						IF GradientToggle THEN
							st_LEDControl.Execute := FALSE;
							SFCStep := 4;
						END_IF
						GradientToggle := NOT GradientToggle;
					END_IF
					
				3: 
					IF NOT animationReady AND NOT LedBusy.Q THEN
							AnimationReady := SetAnimation(ActiveLeds := ui_activeLeds, charging:= getChargingState() = eDCstate.charging, reset := getChargingState() = eDCstate.idle, ledstoAnimate := LedsToAnimate);
					END_IF
					
					IF AnimationReady THEN
						AnimationReady := FALSE;
						st_LEDControl.Execute := NOT st_LEDControl.Execute;
						SFCStep := SFCStep + 1;
					END_IF
				ELSE
					bufferReady := TRUE;
			END_CASE
			
			ton_LEDdataSend(in:= NOT ton_LEDdataSend.Q AND bufferReady);
			IF ton_LEDDataSend.Q THEN
				ReadyToTransmit := TRUE;
			END_IF
			
			IF ReadyToTransmit AND NOT ledbusy.Q THEN
				SFCStep := 0;
				st_LEDControl.UPDATE 	:= NOT st_LEDControl.UPDATE;
				st_LEDControl.Execute 	:= NOT st_LEDControl.execute;	
			END_IF		
	END_CASE
END_IF

METHOD GetChargingState : eDCstate; 
VAR_INPUT
END_VAR
IF machinedata.r_DCCurrent > 10 THEN
	GetChargingState := eDCstate.discharging;
	//b_charging := FALSE;	
	//b_discharging := TRUE;
ELSIF machinedata.r_DCCurrent < -10 THEN
	GetChargingState := eDCstate.charging;
	//b_charging := TRUE;
	//b_discharging := FALSE;
ELSE
	GetChargingState := eDCstate.idle;
	//b_discharging := FALSE;
	//b_charging := FALSE;	
END_IF
END_METHOD

METHOD SetAnimation : BOOL;
VAR_INPUT
	ActiveLeds			: UINT;
	Charging			: BOOL;
	reset				: BOOL;
	LedsToAnimate		: BYTE := 5;	
END_VAR

VAR_INST
	AnimateResetToggle	: BYTE;
	//moveCounter			: CTUD;
	//ready				: BOOL;
	ledcounter			: BYTE;
END_VAR

//movecounter(pv := LedsToAnimate +1);
//moveCounter.LOAD := moveCounter.QD AND Charging;
//moveCounter.Reset := moveCounter.CV > movecounter.PV AND NOT Charging OR Reset;

//CASE AnimateResetToggle OF
//0:		AnimateResetToggle := AnimateResetToggle +1;
//		moveCounter.CU := FALSE;
//		moveCounter.CD := FALSE;
//	ELSE
//		AnimateResetToggle := 0;
//		moveCounter.cu := NOT charging;
//		movecounter.cd := Charging;
//		st_LEDControl.length 	:= 1;
//		st_LEDControl.command	:= 1; //move
//		st_LEDControl.parameter := 0;
//		st_LEDControl.index :=  ui_ActiveLeds + moveCounter.CV -1;
//		SetAnimation := TRUE;
//END_CASE

IF NOT RESET THEN
	ledcounter := ledcounter + SEL(charging,1 ,-1);
	IF ledcounter >= LedsToAnimate * 2 OR ledcounter = 0 THEN
		ledcounter := SEL(charging,0 ,LedsToAnimate * 2);	 
	END_IF
	
	st_LEDControl.length 	:= 1;
	st_LEDControl.command	:= 1; //move
	st_LEDControl.parameter := 
	st_LEDControl.index :=  ActiveLeds + ledcounter/2;
ELSE
	ledcounter := 0;
END_IF

SetAnimation := TRUE;
END_METHOD

METHOD SetColor : LEDColor

VAR_INPUT
	Brightness		: BYTE;
END_VAR

VAR
	tempColorValue	: USINT;
END_VAR
CASE machinedata.e_systemStatus OF
	eSystemStatus.neutral: 		
		SetColor.blue	:= Brightness;
		SetColor.red	:= Brightness;
		SetColor.green	:= Brightness;

	eSystemStatus.normal: 
		SetColor.blue	:= 0;
		SetColor.red	:= 0;
		SetColor.green	:= Brightness;
	
	eSystemStatus.attention: 
		SetColor.blue	:= Brightness;
		SetColor.red	:= 0;
		SetColor.green	:= 0;
	eSystemStatus.warning: //yelow
		SetColor.blue	:= 0;
		SetColor.red	:= Brightness;
		SetColor.green	:= Brightness/3;
	
	eSystemStatus.error: 
		SetColor.blue	:= 0;
		SetColor.red	:= Brightness;
		SetColor.green	:= 0;	
END_CASE

//Change RGB order
IF st_params.ColorOrder = eColorOrder.GRB THEN
	tempColorValue := setColor.Red;
	setcolor.red := setcolor.green;
	SetColor.green := tempColorValue;
END_IF
END_METHOD

END_FUNCTION_BLOCK

// ---- POUs/Objects/Enclosure/Climate/FB_EnclosureClimate.TcPOU
FUNCTION_BLOCK FB_EnclosureClimate
VAR_IN_OUT CONSTANT
	st_params				: ST_EnclosureClimate_params;
END_VAR
VAR_OUTPUT
	get						: ST_EnclosureClimate_get;
END_VAR

VAR
	TempRead		AT %I* : ST_AnalogInputData;
	HumRead			AT %I* : ST_AnalogInputData;
	
	scaleTemp				: FB_CTRL_SCALE;
	scaleHum				: FB_CTRL_SCALE;
	scaleParams				: ST_CTRL_SCALE_Params;
END_VAR

scaleParams.tCtrlCycleTime := T#100MS;
	scaleParams.tTaskCycleTime := T#1MS;
	scaleParams.fInMax := 16#7FFF;
	scaleParams.fInMin := 16#0000;
	scaleParams.fOutMax := 60;
	scaleParams.fOutMin:= -40;

scaleTemp(fin := TempRead.Value, fout => get.r_Temperature, stParams := scaleParams);
scaleParams.fOutMax := 100;
scaleParams.fOutMin := 0;
scaleHum(fin := HumRead.Value, fout => get.r_Humidity, stParams := scaleParams);

METHOD PUBLIC GetDiagnostics
VAR_IN_OUT
	AddError		: ARRAY [*] OF FB_AddErrorST;
	a_ActiveEvents	: ARRAY [*] OF ST_ErrorStruct;
	w_Index			: WORD;
END_VAR


VAR
	by_errCt	: BYTE;
	by_warnCt	: BYTE;
END_VAR
	(*Humidity High*)		AddError[w_Index](
		b_ErrorTrig			:= get.events.b_HumidityHigh,
		out_ST_Error			:= a_ActiveEvents[w_Index],
		w_ErrorID					:= 1,
		e_ObjectID				:=  eObject_ID.Enclosure_climate,
		s_Message				:= 'humidity high',
		e_sev					:= eseverity.Warning,
		b_AutoClear			:= TRUE
		);
		w_Index := w_Index +1;
	
	(*Humidity Too High*)		AddError[w_Index](
		b_ErrorTrig			:= get.events.b_HumidityTooHigh,
		out_ST_Error			:= a_ActiveEvents[w_Index],
		w_ErrorID					:= 2,
		s_Message				:= 'humidity too high',
		e_sev					:= eseverity.QuickShutdown,
		e_ErrAckAccess		:= eErrAckAccess.Operator
	);
	w_Index := w_Index +1;
	
	(*Temperature High*)		AddError[w_Index](
		b_ErrorTrig			:= get.events.b_TemperatureHigh,
		out_ST_Error			:= a_ActiveEvents[w_Index],
		w_ErrorID					:= 3,
		s_Message				:= 'temperature high',
		e_sev					:= eseverity.warning,
		b_AutoClear			:= TRUE
	);
	w_Index := w_Index +1;
	
	(*Temperature Too High*)	AddError[w_Index](
		b_ErrorTrig			:= get.events.b_TemperatureTooHigh,
		out_ST_Error			:= a_ActiveEvents[w_Index],
		w_ErrorID					:= 4,
		s_Message				:= 'temperature too high',
		e_sev					:= eseverity.Quickshutdown,
		e_ErrAckAccess		:= eErrAckAccess.Operator
	);

	w_Index := w_Index +1;
	
	(*Temperature Low*)	AddError[w_Index](
		b_ErrorTrig			:= get.events.b_TemperatureLow,
		out_ST_Error			:= a_ActiveEvents[w_Index],
		w_ErrorID					:= 5,
		s_Message				:= 'temperature low',
		e_sev					:= eseverity.Warning,
		b_AutoClear			:= TRUE
	);
	w_Index := w_Index +1;
	
	(*Temperature Too Low*)	AddError[w_Index](
		b_ErrorTrig			:= get.events.b_TemperatureTooLow,
		out_ST_Error			:= a_ActiveEvents[w_Index],
		w_ErrorID					:= 6,
		s_Message				:= 'temperature too low',
		e_sev					:= eseverity.Normalshutdown,
		e_ErrAckAccess		:= eErrAckAccess.Operator
	);
	w_Index := w_Index +1;
	
	(*4-20ma Overrange*)	AddError[w_Index](
		b_ErrorTrig			:= get.events.b_AIOverrange,
		out_ST_Error			:= a_ActiveEvents[w_Index],
		w_ErrorID					:= 7,
		s_Message				:= 'analog input temp/humid overrange',
		e_sev					:= eseverity.Warning,
		b_AutoClear			:= TRUE
	);
	w_Index := w_Index +1;
	
	(*4-20ma Underrange*)	AddError[w_Index](
		b_ErrorTrig			:= get.events.b_AIUnderrange,
		out_ST_Error			:= a_ActiveEvents[w_Index],
		w_ErrorID					:= 8,
		s_Message				:= 'analog input temp/humid underrange',
		e_sev					:= eseverity.Warning,
		b_AutoClear			:= TRUE
	);
	w_Index := w_Index +1;
	
	(*Analog input error*)	AddError[w_Index](
		b_ErrorTrig			:= get.events.b_AIError,
		out_ST_Error			:= a_ActiveEvents[w_Index],
		w_ErrorID					:= 9,
		s_Message				:= 'analog input temp/humid error',
		e_sev					:= eseverity.warning,
		b_AutoClear			:= TRUE
	);
	w_Index := w_Index +1;
	
	(*Analog input error*)	AddError[w_Index](
		b_ErrorTrig				:= get.events.b_DewpointTooHigh,
		out_ST_Error			:= a_ActiveEvents[w_Index],
		w_ErrorID				:= 10,
		s_Message				:= 'dewpoint too high alarm',
		e_sev					:= eseverity.normalshutdown,
	);
	w_Index := w_Index +1;
END_METHOD

METHOD PRIVATE SetEvents : BOOL
VAR_IN_OUT
	get : ST_EnclosureClimate_get;
	st_params : ST_EnclosureClimate_params;
END_VAR

VAR_INST
	sr_HumHigh			: SR;
	sr_HumTooHigh		: SR;
	sr_TempHigh			: SR;
	sr_TempTooHigh		: SR;
	sr_TempLow			: SR;
	sr_TempTooLow		: SR;
END_VAR
//set events
get.events.b_AIError := TempRead.Status.Error OR HumRead.Status.Error;
get.events.b_AIUnderrange := TempRead.Status.Underrange OR HumRead.Status.Underrange;
get.events.b_AIOverrange := TempRead.Status.Overrange OR HumRead.Status.Overrange;

sr_HumHigh(
	SET1:= get.r_Humidity > st_params.r_HumidityHigh, 
	RESET:= get.r_Humidity <= st_params.r_HumidityHigh - st_params.r_HumidityHysteris,
	Q1 => get.events.b_HumidityHigh);
sr_HumTooHigh(
	SET1:= get.r_Humidity > st_params.r_HumidityTooHigh, 
	RESET:= get.r_Humidity <= st_params.r_HumidityTooHigh - st_params.r_HumidityHysteris,
	Q1 => get.events.b_HumidityTooHigh);	
sr_TempHigh(
	SET1:= get.r_Temperature > st_params.r_TemperatureHigh, 
	RESET:= get.r_Temperature <= st_params.r_TemperatureHigh - st_params.r_TemperatureHysteris,
	Q1 => get.events.b_TemperatureHigh);	
sr_TempTooHigh(
	SET1:= get.r_Temperature > st_params.r_TemperatureTooHigh, 
	RESET:= get.r_Temperature <= st_params.r_TemperatureTooHigh - st_params.r_TemperatureHysteris,
	Q1 => get.events.b_TemperatureTooHigh);
sr_TempLow(
	SET1:= get.r_Temperature < st_params.r_TemperatureLow, 
	RESET:= get.r_Temperature >= st_params.r_TemperatureLow + st_params.r_TemperatureHysteris,
	Q1 => get.events.b_TemperatureLow);
sr_TempTooLow(
	SET1:= get.r_Temperature < st_params.r_TemperatureTooLow, 
	RESET:= get.r_Temperature >= st_params.r_TemperatureTooLow + st_params.r_TemperatureHysteris,
	Q1 => get.events.b_TemperatureTooLow);
END_METHOD

END_FUNCTION_BLOCK

// ---- POUs/Objects/Enclosure/Doors/FB_DoorsNLocks.TcPOU
FUNCTION_BLOCK FB_DoorsNLocks
VAR_OUTPUT
	get 		: ST_DoorsNLocks_get;
END_VAR

VAR
	b_ControlPanelDoorfb	AT %I* : BOOL;
	b_ClientPanelDoorfb		AT %I* : BOOL;
END_VAR

get.b_ControlPanelDoorClosed := b_ControlPanelDoorfb;
get.b_ClientpanelDoorClosed	:= b_ClientPanelDoorfb;

METHOD PUBLIC GetDiagnostics
VAR_IN_OUT
	AddError		: ARRAY [*] OF FB_AddErrorST;
	a_ActiveEvents	: ARRAY [*] OF ST_ErrorStruct;
	w_Index			: WORD;
END_VAR

VAR_OUTPUT
	b_errorActive	: BOOL;
	b_warningActive	: BOOL;
END_VAR

VAR
	by_errCt	: BYTE;
	by_warnCt	: BYTE;
END_VAR
	(*Client door open*)		AddError[w_Index](
		b_ErrorTrig			:= NOT(get.b_ClientpanelDoorClosed),
		out_ST_Error			:= a_ActiveEvents[w_Index],
		w_ErrorID					:= 1,
		e_ObjectID				:=  eObject_ID.Enclosure_doors,
		s_Message				:= 'client panel opened',
		e_sev					:= eseverity.info,
		b_AutoClear			:= TRUE
		);
		w_Index := w_Index +1;
		
	(*Client door open*)		AddError[w_Index](
		b_ErrorTrig			:= NOT(get.b_ControlPanelDoorClosed),
		out_ST_Error			:= a_ActiveEvents[w_Index],
		w_ErrorID					:= 2,
		s_Message				:= 'control panel opened',
		e_sev					:= eseverity.info,
		b_AutoClear			:= TRUE
		);
		w_Index := w_Index +1;
END_METHOD

END_FUNCTION_BLOCK

// ---- POUs/Objects/PLCStatus/FB_PLCState.TcPOU
FUNCTION_BLOCK FB_PLCState
VAR_OUTPUT
	EL9410					AT %I* : ST_EL9410;
	get							: ST_PLCstate_get;
END_VAR
VAR
	ton_refreshpulse					: TON := (PT := T#500ms);
	events : ST_PLC_events;
	by_PNErrorsAllowed					: BYTE;
	ui_EthercatMasterState		AT %I* : UINT;
	ui_ProfinetNoErrorDevices	AT %I* : UINT;
	ui_ProfinetNoDiagDevices	AT %I* : UINT;
	ui_SafetyLogicState			AT %I* : UINT;	
	
	ton_SystemReady					: TON := (IN := FALSE, PT := T#15S);	
	
	fb_cpuload 						: TC_CpuUsage;
	
END_VAR

events.b_EthercatMasterFault := ui_EthercatMasterState <> 0;

ton_SystemReady(IN:= TRUE);
GVL.b_SystemReady	:= ton_SystemReady.Q;

IF settings.Configuration.e_PNcouplerType = 0 THEN
	by_PNErrorsAllowed := 3;
ELSE 
	by_PNErrorsAllowed := 2;
END_IF

// get cpu load
ton_refreshpulse(IN := NOT ton_refreshpulse.Q);
fb_cpuload(start:= ton_refreshpulse.Q,
	TMOUT:= T#5S);
get.r_CPUload:= TO_REAL(fb_cpuload.USAGE);

IF ui_ProfinetNoErrorDevices > by_PNErrorsAllowed THEN
	get.e_ProfinetState := eNetcomState.Error;
ELSIF ui_ProfinetNoDiagDevices > by_PNErrorsAllowed THEN
	get.e_ProfinetState := eNetcomState.Warning;
ELSIF ui_ProfinetNoErrorDevices <= by_PNErrorsAllowed AND ui_ProfinetNoDiagDevices <= by_PNErrorsAllowed THEN
	get.e_ProfinetState := eNetcomState.OK;
ELSE
	get.e_ProfinetState := eNetcomState.NotConnected;
END_IF

IF ui_EthercatMasterState = 0 THEN
	get.e_EthercatState := eNetcomState.OK;
ELSIF ui_EthercatMasterState = 1 THEN
	get.e_EthercatState := eNetcomState.NotConnected;
ELSE
	get.e_EthercatState := eNetcomState.Error;
END_IF

METHOD GetDiagnostics
VAR_IN_OUT
	AddError		: ARRAY [*] OF FB_AddErrorST;
	a_ActiveEvents	: ARRAY [*] OF ST_ErrorStruct;
	w_Index			: WORD;
END_VAR
(*PLC io supply fault*)		AddError[w_Index](
					b_ErrorTrig			:= EL9410.bit_UpUndervoltage OR EL9410.bit_UsUndervoltage,
					out_ST_Error			:= a_ActiveEvents[w_Index],
					w_ErrorID					:= 1,
					e_ObjectID				:= eObject_ID.PLC,
					s_Message				:= 'EL9410 supply fault',
					e_sev					:= eSeverity.Quickshutdown
				);
				w_Index := w_Index +1;
				
(*Ethercat master fault*)		AddError[w_Index](
					b_ErrorTrig			:= events.b_EthercatMasterFault,
					out_ST_Error			:= a_ActiveEvents[w_Index],
					w_ErrorID					:= 2,
					s_Message				:= 'Ethercat master fault',
					e_sev					:= eSeverity.normalshutdown,
				);
				w_Index := w_Index +1;
END_METHOD

END_FUNCTION_BLOCK

// ---- POUs/Objects/PeakshaveBox/FB_PeakshaveBox.TcPOU
FUNCTION_BLOCK FB_PeakshaveBox
VAR_IN_OUT CONSTANT
	st_params 			: ST_peakshavebox_params;
END_VAR

VAR_INPUT
	set					: ST_peakshaveBox_set;
END_VAR

VAR_OUTPUT
	get					: ST_PeakshaveBox_get; 
END_VAR

VAR
	EmptyGet				: ST_PeakshaveBox_get;
	WagoBus					: FB_Wago750354_Buscoupler;
	WagoPQ					: FB_Wago750495_PowerMonitor;
	BeckhoffBus				: FB_EK1100;
	BeckhoffPQ				: FB_EL3453;

	ton_activationDelay		: TON := (PT := T#2S);
END_VAR

VAR_INPUT
	b_enable			: BOOL;
END_VAR

VAR PERSISTENT
	b_BreakerControl 			: BOOL;
	ui_CtRange		 			: UINT := 1000;
	r_VTRatio		 			: REAL := 1;
	b_InverseCTdirection		: BOOL;
END_VAR

ton_activationDelay(IN := get.b_dataOK AND b_enable AND get.b_buscouplerReady, Q => get.b_active);// AND NOT Powermonitor.get.StatusWord.b_Error;
//Instantiate FBs

//PSB settings can only be updated when not active
IF NOT b_enable THEN
	 b_breakerControl := set.b_BreakerControl;
	 ui_ctrange := set.ui_CtRange;
	 r_vtRatio := set.r_VTRatio;
	 b_inverseCTdirection := set.b_InverseCTdirection;
END_IF

get.b_SettingsChangePending := 	(b_breakerControl <> set.b_BreakerControl) OR 
								(ui_ctrange <> set.ui_CtRange) OR 
								(r_vtRatio <> set.r_VTRatio) OR 
								(b_inverseCTdirection <> set.b_InverseCTdirection);
 
CASE st_params.PSBhardware OF
	ePSBHardware.Wago: 
		get.b_dataOK := AcCheck(get.Powermonitor.ar_LineVoltage[0] ,get.Powermonitor.ar_Frequency[0]);
		WagoBus();
		WagoPQ(b_enable:= WagoBus.get.b_SlaveReady, Fastmode := st_params.fastmode, CTinverse := b_InverseCTdirection);
		MapWago();
	ePSBhardware.Beckhoff:
		BeckhoffBus();
		BeckhoffPQ(VoltageRatio := r_VTRatio, CurrentRatio := UINT_TO_INT(ui_CtRange), CTinverse := b_InverseCTdirection);
		MapBeckhoff();	
END_CASE


IF get.b_active THEN
	get.PSBmode := ePSBMode.Monitor;
	IF b_BreakerControl THEN
		get.PSBmode := ePSBMode.MonitorControl;
	END_IF
ELSE
	get.PSBmode := ePSBMode.None;
END_IF

METHOD PUBLIC GetDiagnostics
VAR_IN_OUT
	AddError		: ARRAY [*] OF FB_AddErrorST;
	a_ActiveEvents	: ARRAY [*] OF ST_ErrorStruct;
	w_Index			: WORD;
END_VAR
(*Voltage L1 fault*) 	AddError[w_Index](
			b_ErrorTrig			:= NOT Get.b_buscouplerReady AND b_enable,
			out_ST_Error			:= a_ActiveEvents[w_Index],
			w_ErrorID				:= 1,
			e_ObjectID				:= eObject_ID.PeakshaveBox,
			s_Message				:= 'Buscoupler not detected',
			e_sev					:= eseverity.Warning,
			b_autoClear				:= TRUE
			);
		w_Index := w_Index +1;


(*Voltage L1 fault*) 	AddError[w_Index](
			b_ErrorTrig			:= Get.Powerstatus.b_Error_Phase[1],
			out_ST_Error			:= a_ActiveEvents[w_Index],
			w_ErrorID				:= 2,
			e_ObjectID				:= eObject_ID.PeakshaveBox,
			s_Message				:= 'L1 error',
			e_sev					:= eseverity.Warning,
			b_autoClear				:= TRUE
			);
		w_Index := w_Index +1;
		
(*Voltage L2 fault*) 	AddError[w_Index](
			b_ErrorTrig			:= Get.Powerstatus.b_Error_Phase[2],
			out_ST_Error			:= a_ActiveEvents[w_Index],
			w_ErrorID				:= 3,
			e_ObjectID				:= eObject_ID.PeakshaveBox,
			s_Message				:= 'L2 error',
			e_sev					:= eseverity.Warning,
			b_autoClear				:= TRUE
			);
		w_Index := w_Index +1;
		
(*Voltage L3 fault*) 	AddError[w_Index](
			b_ErrorTrig			:= Get.Powerstatus.b_Error_Phase[3],
			out_ST_Error			:= a_ActiveEvents[w_Index],
			w_ErrorID				:= 4,
			e_ObjectID				:= eObject_ID.PeakshaveBox,
			s_Message				:= 'L3 error',
			e_sev					:= eseverity.Warning,
			b_autoClear				:= TRUE
			);
		w_Index := w_Index +1;
		
(*Powermonitor current L1 out of range*) 	AddError[w_Index](
			b_ErrorTrig			:= Get.PowerStatus.b_OverCurrent AND Get.PowerStatus.b_Error_Phase[1],
			out_ST_Error			:= a_ActiveEvents[w_Index],
			w_ErrorID				:= 6,
			e_ObjectID				:= eObject_ID.PeakshaveBox,
			s_Message				:= 'Powermonitor current L1 out of range',
			e_sev					:= eseverity.Warning,
			b_autoClear				:= TRUE
			);
		w_Index := w_Index +1;
		
(*Powermonitor current L2 out of range*) 	AddError[w_Index](
			b_ErrorTrig			:= Get.PowerStatus.b_OverCurrent AND Get.PowerStatus.b_Error_Phase[2],
			out_ST_Error			:= a_ActiveEvents[w_Index],
			w_ErrorID				:= 7,
			e_ObjectID				:= eObject_ID.PeakshaveBox,
			s_Message				:= 'Powermonitor current L2 out of range',
			e_sev					:= eseverity.Warning,
			b_autoClear				:= TRUE
			);
		w_Index := w_Index +1;
		
(*Powermonitor current L3 out of range*) 	AddError[w_Index](
			b_ErrorTrig			:= Get.PowerStatus.b_OverCurrent AND Get.PowerStatus.b_Error_Phase[3],
			out_ST_Error			:= a_ActiveEvents[w_Index],
			w_ErrorID				:= 8,
			e_ObjectID				:= eObject_ID.PeakshaveBox,
			s_Message				:= 'Powermonitor current L3 out of range',
			e_sev					:= eseverity.Warning,
			b_autoClear				:= TRUE
			);
		w_Index := w_Index +1;
		
(*Powermonitor general warning*) 	AddError[w_Index](
			b_ErrorTrig			:= Get.PowerStatus.b_GeneralWarning,
			out_ST_Error			:= a_ActiveEvents[w_Index],
			w_ErrorID				:= 9,
			e_ObjectID				:= eObject_ID.PeakshaveBox,
			s_Message				:= 'Powermonitor general warning',
			e_sev					:= eseverity.Warning,
			b_autoClear				:= TRUE
			);
		w_Index := w_Index +1;
		

		
(*Powermonitor overcurrent fault*) 	AddError[w_Index](
			b_ErrorTrig				:= Get.PowerStatus.b_OverCurrent,
			out_ST_Error			:= a_ActiveEvents[w_Index],
			w_ErrorID				:= 11,
			e_ObjectID				:= eObject_ID.PeakshaveBox,
			s_Message				:= 'Powermonitor overcurrent fault',
			e_sev					:= eseverity.Warning,
			b_autoClear				:= TRUE
			);
		w_Index := w_Index +1;
		
(*Powermonitor overvoltage fault*) 	AddError[w_Index](
			b_ErrorTrig				:= Get.PowerStatus.b_OverVoltage,
			out_ST_Error			:= a_ActiveEvents[w_Index],
			w_ErrorID				:= 12,
			e_ObjectID				:= eObject_ID.PeakshaveBox,
			s_Message				:= 'Powermonitor overvoltage fault',
			e_sev					:= eseverity.Warning,
			b_autoClear				:= TRUE
			);
		w_Index := w_Index +1;
		
(*Powermonitor undervoltage fault*) 	AddError[w_Index](
			b_ErrorTrig				:= Get.PowerStatus.b_UnderVoltage,
			out_ST_Error			:= a_ActiveEvents[w_Index],
			w_ErrorID				:= 13,
			e_ObjectID				:= eObject_ID.PeakshaveBox,
			s_Message				:= 'Powermonitor undervoltage fault',
			e_sev					:= eseverity.Warning,
			b_autoClear				:= TRUE
			);
		w_Index := w_Index +1;

	
	(*Setting change pending*) 	AddError[w_Index](
			b_ErrorTrig				:= get.b_SettingsChangePending,
			out_ST_Error			:= a_ActiveEvents[w_Index],
			w_ErrorID				:= 14,
			e_ObjectID				:= eObject_ID.PeakshaveBox,
			s_Message				:= 'PSB settings change blocked, disable PSB to apply',
			e_sev					:= eseverity.Warning,
			b_autoClear				:= TRUE
			);
		w_Index := w_Index +1;
END_METHOD

METHOD MapBeckhoff : BOOL

VAR
	i : INT;
END_VAR

VAR_INST
	voltageOK : BOOL;
	currentOK : BOOL;
	PhaseError: BOOL;
END_VAR
get.b_buscouplerReady := beckhoffbus.state = 8 AND beckhoffpq.ui_EL3443BoxState = 8;

IF NOT get.b_buscouplerReady THEN
	get := EmptyGet;	
ELSE
	get.powermonitor.ar_ActivePower := beckhoffPQ.r_ActivePower;
	get.Powermonitor.ar_ApparentPower := beckhoffPQ.r_ApparentPower;
	get.Powermonitor.ar_ReactivePower := beckhoffPQ.r_ReactivePower;
	get.Powermonitor.ar_Current := beckhoffPQ.r_Current;
	get.Powermonitor.ar_LineVoltage := beckhoffPQ.r_LineVoltage;
	get.Powermonitor.ar_PhaseVoltage := beckhoffPQ.r_PhaseVoltage;
	get.powermonitor.ar_Frequency := beckhoffPQ.r_Frequency;
	get.Powermonitor.li_TimeVoltZeroCrossup := beckhoffPQ.li_TimeVoltZeroCrossup;
	//get.Powermonitor.ar_THD := beckhoffPQ
	get.Powermonitor.r_EnergyConsumed := beckhoffPQ.r_ActiveEnergyConsumed;
	get.Powermonitor.r_EnergySupplied:= beckhoffPQ.r_ActiveEnergySupplied;
	get.Powermonitor.r_VoltageUnbalance := beckhoffPQ.r_VoltageUnbalance;
	get.Powermonitor.r_CurrentUnbalance := beckhoffPQ.r_CurrentUnbalance;
	get.Powermonitor.ar_PowerFactor := beckhoffPQ.r_PowerFactor;
	
	get.PowerStatus.b_RotaryField := beckhoffPQ.TotalStatus.bit_GridDirection;
	IF beckhoffPQ.TotalStatus.bit_FrequencyGuardError THEN
		get.Powermonitor.e_ACrotationStatus := eAcrotationstate.None;
	ELSIF beckhoffPQ.TotalStatus.bit_GridDirection THEN
		get.Powermonitor.e_ACrotationStatus := eAcrotationstate.Right;
	ELSE
		get.Powermonitor.e_ACrotationStatus := eAcrotationstate.Left;
	END_IF
	
	
	
	voltageOK := beckhoffPQ.r_LineVoltage[0] <> 0;
	get.PowerStatus.b_OverCurrent := FALSE;
	get.PowerStatus.b_OverVoltage := FALSE;
	get.PowerStatus.b_UnderVoltage := FALSE;
	get.PowerStatus.b_GeneralWarning := 
		beckhoffPQ.TotalStatus.bit_ActivePowerGuardWarning OR
		beckhoffPQ.TotalStatus.bit_ApparentPowerGuardWarning OR
		beckhoffPQ.TotalStatus.bit_FrequencyGuardwarning OR
		beckhoffPQ.TotalStatus.bit_NeutralCurrentGuardWarning OR
		beckhoffPQ.TotalStatus.bit_PowerQualityGuardWarning AND get.b_buscouplerReady;
	get.PowerStatus.b_GeneralFault := 
		beckhoffPQ.TotalStatus.bit_ActivePowerGuardError OR
		beckhoffPQ.TotalStatus.bit_ApparentPowerGuardError OR
		beckhoffPQ.TotalStatus.bit_FrequencyGuardError OR
		beckhoffPQ.TotalStatus.bit_NeutralCurrentGuardError OR
		beckhoffPQ.TotalStatus.bit_PowerQualityGuardError OR
		NOT beckhoffPQ.TotalStatus.bit_SystemState AND get.b_buscouplerReady;
		
	
	//loop through phases 
	FOR i := 1 TO 3 DO
		PhaseError := FALSE;
		CurrentOK := TRUE;
		
		IF beckhoffpq.PhaseStatus[i].bit_VoltageGuardError THEN  
			get.PowerStatus.b_UnderVoltage := TRUE;
			voltageOK := FALSE;	
			PhaseError := TRUE;
		END_IF
		
		IF beckhoffpq.PhaseStatus[i].bit_InaccurateVoltage THEN  
			voltageOK := FALSE;	
			PhaseError := TRUE;
		END_IF
		
		IF beckhoffpq.PhaseStatus[i].bit_Overvoltage THEN
			get.PowerStatus.b_OverVoltage := TRUE;
			voltageOK := FALSE;	
			PhaseError := TRUE;
		END_IF
		
		IF beckhoffpq.PhaseStatus[i].bit_Overcurrent THEN  
			CurrentOK := FALSE;	
			PhaseError := TRUE;
		END_IF
		
		IF beckhoffpq.PhaseStatus[i].bit_Overcurrent THEN
			get.PowerStatus.b_OverCurrent := TRUE;
			CurrentOK := FALSE;
			PhaseError := TRUE;
		END_IF
		
		IF beckhoffPq.PhaseStatus[i].bit_VoltageGuardWarning OR beckhoffPq.PhaseStatus[i].bit_CurrentGuardWarning THEN
			get.PowerStatus.b_GeneralWarning := TRUE;
		END_IF
			
		IF beckhoffPq.PhaseStatus[i].bit_VoltageGuardError OR beckhoffPq.PhaseStatus[i].bit_CurrentGuardError THEN
			get.PowerStatus.b_GeneralFault := TRUE;
			PhaseError := TRUE;
		END_IF
			
		get.PowerStatus.b_Error_Phase[i] := PhaseError;
	END_FOR
	
	get.b_dataOK := VoltageOK AND currentOK AND beckhoffPQ.TotalStatus.bit_SystemState;
END_IF
END_METHOD

METHOD MapWago : BOOL
VAR_INPUT
END_VAR
get.b_buscouplerReady := wagobus.get.b_SlaveReady;

IF NOT get.b_buscouplerReady THEN
	get := EmptyGet;	
ELSE
	get.Powermonitor.ar_ActivePower := WagoPQ.get.Data.ar_ActivePower;
	get.Powermonitor.ar_ReactivePower := WagoPQ.get.Data.ar_ReactivePower;
	get.Powermonitor.ar_ApparentPower := WagoPQ.get.Data.ar_ApparentPower;
	get.Powermonitor.ar_Current := WagoPQ.get.Data.ar_CurrentRMS;
	get.Powermonitor.ar_LineVoltage := WagoPQ.get.Data.ar_VoltageLL;
	get.Powermonitor.ar_PhaseVoltage := WagoPQ.get.Data.ar_VoltageLN;
	get.powermonitor.ar_Frequency := WagoPQ.get.Data.ar_Frequency;
	//get.Powermonitor.ar_THD := beckhoffPQ
	get.Powermonitor.r_EnergyConsumed := WagoPQ.get.Data.r_ActiveEnergyImport;
	get.Powermonitor.r_EnergySupplied:= WagoPQ.get.Data.r_ActiveEnergyExport;
	get.Powermonitor.r_VoltageUnbalance := 0;
	get.Powermonitor.r_CurrentUnbalance := 0;
	get.Powermonitor.ar_PowerFactor := wagoPQ.get.Data.ar_Powerfactor;
	
	get.PowerStatus.b_Error_Phase[1] := wagoPQ.get.StatusWord.b_Error_L1;
	get.PowerStatus.b_Error_Phase[2] := wagoPQ.get.StatusWord.b_Error_L2;
	get.PowerStatus.b_Error_Phase[3] := wagoPQ.get.StatusWord.b_Error_L3;
	get.PowerStatus.b_OverCurrent := wagoPQ.get.ExtStatusWord.b_OverCurrent;
	get.PowerStatus.b_OverVoltage := wagoPQ.get.ExtStatusWord.b_OverVoltage;
	get.PowerStatus.b_RotaryField := wagoPQ.get.ExtStatusWord.b_RotaryField;
	get.PowerStatus.b_GeneralFault := wagoPQ.get.StatusWord.b_Error;
	get.PowerStatus.b_GeneralWarning := wagoPQ.get.StatusWord.b_Warning;
	
	IF get.PowerStatus.b_GeneralFault THEN
		get.Powermonitor.e_ACrotationStatus := eAcrotationstate.None;
	ELSIF beckhoffPQ.TotalStatus.bit_GridDirection THEN
		get.Powermonitor.e_ACrotationStatus := eAcrotationstate.Right;
	ELSE
		get.Powermonitor.e_ACrotationStatus := eAcrotationstate.Left;
	END_IF
END_IF
END_METHOD

END_FUNCTION_BLOCK

// ---- POUs/Functions-FBs-Programs/IO_modules/Wago/FB_Wago750354_BusCoupler.TcPOU
FUNCTION_BLOCK INTERNAL FB_Wago750354_BusCoupler
VAR_INPUT
//	b_KbusCycleOverrunFlagDisable			AT %Q* : BOOL;
//	b_InputProcessDataHoldRequest			AT %Q* : BOOL;
//	b_OutputProcessDataHoldRequest			AT %Q* : BOOL;
//	b_OutputDataClearRequest				AT %Q* : BOOL;
	
	b_AckDiagnostics						: BOOL;
	b_ClearDiagnostics						: BOOL;
END_VAR
VAR_OUTPUT
//	b_kBusCycleOverRun						AT %I* : BOOL;
//	b_InputProcessDataHoldAck				AT %I* : BOOL;
//	b_OutputProcessDataHoldAck				AT %I* : BOOL;
//	b_OutputProcessDataClearAck				AT %I* : BOOL;
//	b_NewMessageAvailable					AT %I* : BOOL;
	get											  : ST_Wago750354_get;
END_VAR
VAR	
	ui_DiagnosticsStatusWord			AT %I* : UINT;
	ui_State							AT %I* : UINT;
	DiagnosticsControlWord				AT %Q* : UINT;
END_VAR

get.b_SlaveReady := ui_State = 8;

END_FUNCTION_BLOCK

// ---- POUs/Functions-FBs-Programs/IO_modules/Wago/FB_Wago750495_PowerMonitor.TcPOU
FUNCTION_BLOCK INTERNAL FB_Wago750495_PowerMonitor

VAR
	a_DataIN				AT %I* : ARRAY[1..24] OF USINT;
	a_DataOUT				AT %Q* : ARRAY[1..8] OF USINT;
	set						: ST_Wago750495_Set;	
	emptydata				: ST_Wago750495_Get;		
END_VAR

VAR_INPUT
	b_Enable				: BOOL;
	CTinverse				: BOOL;
	Fastmode				: BOOL;
END_VAR

VAR_OUTPUT
	get						: ST_Wago750495_Get;
END_VAR

//Check if changes 

//write control word and recieve answer
WriteReadRequest(get:= get, b_enable:= b_Enable, fastmode := fastmode);

// Every 1s stat data
ReadStatData(statusword := get.StatusWord,
			ExtStatusWord := get.ExtStatusWord);

IF NOT b_enable THEN
	get := emptydata;
END_IF

METHOD PRIVATE ReadStatData : BOOL
VAR_IN_OUT
	statusword		: ST_Wago750495_StatusWord;
	ExtStatusWord	: ST_Wago750495_ExtStatusWord;
END_VAR

VAR_INST
	ton_RefreshRate		: TON :=(PT := T#500MS);	
	usi_stat_sel		: USINT;
END_VAR
ton_RefreshRate(IN := NOT ton_RefreshRate.Q);
IF ton_RefreshRate.Q THEN
	//StatusWord byte 0
	statusword.b_Error_L1 := a_DataIN[1].0;
	statusword.b_Error_L2 := a_DataIN[1].1;
	statusword.b_Error_L3 := a_DataIN[1].2;
	statusword.b_Error_IO := a_DataIN[1].3;
	statusword.b_Error := a_DataIN[1].6;
	statusword.b_ComFb := a_DataIN[1].7;
	
	//StatusWord byte 1
	CASE (a_DataIN[2] MOD 4) OF 
		0: Statusword.e_StatIDfb := eWago750495_StatDataID.Phase1;
		1: Statusword.e_StatIDfb := eWago750495_StatDataID.Phase2;
		2: Statusword.e_StatIDfb := eWago750495_StatDataID.Phase3;
		3: Statusword.e_StatIDfb := eWago750495_StatDataID.IOmodule;
	END_CASE
	Statusword.b_Over_4 := a_DataIN[2].2;
	Statusword.b_Over_3 := a_DataIN[2].3;
	Statusword.b_Over_2 := a_DataIN[2].4;	
	Statusword.b_Over_1 := a_DataIN[2].5;
	Statusword.b_Cal := a_DataIN[2].6;
	Statusword.b_Warning := a_DataIN[2].7;
END_IF
END_METHOD

METHOD PRIVATE WriteIOCall : USINT;
VAR_INPUT
	ID1_RQ				: USINT;
	ID2_RQ				: USINT;
	ID3_RQ				: USINT;
	ID4_RQ				: USINT;
	COL_RQ				: USINT;
	r_scale				: REAL;
	r_offset			: REAL;
END_VAR

VAR_OUTPUT
	b_error		: BOOL;
	b_next		: BOOL;
END_VAR

VAR_IN_OUT
	r_out1	: REAL;
	r_out2	: REAL;
	r_out3	: REAL;
	r_out4	: REAL;
END_VAR

VAR_INST
	i_RetryCount	: INT;
	i_cycleCount	: INT;
	a_rDataOut		: ARRAY [1..4] OF REAL;
	ton_Error		: TON := (PT:=T#5S);
	ton_RequestTimer: TON := (PT:=T#2MS);
END_VAR

VAR
	i_MaxRetries	: INT := 30;
	di_Data			: DINT;
	i_int			: INT; 
END_VAR
ton_Error();
ton_RequestTimer(IN:= NOT ton_RequestTimer.Q);

b_next	:= FALSE;
a_dataOUT[4] := COL_RQ;
a_dataOUT[5] := ID1_RQ;
a_dataOUT[6] := ID2_RQ;
a_dataOUT[7] := ID3_RQ;
a_dataOUT[8] := ID4_RQ;

IF ton_RequestTimer.Q AND a_dataOUT[4] = a_dataIN[4] THEN
		IF a_dataIN[5] =  a_dataOUT[5] AND a_dataIN[6] =  a_dataOUT[6] AND a_dataIN[7] =  a_dataOUT[7] AND a_dataIN[8] =  a_dataOUT[8] THEN
			FOR i_int := 1 TO 4 DO
				di_Data:=  SHL(SHL(SHL(a_DataIN[8+4*i_int],8) OR a_DataIN[7+4*i_int],8) OR a_DataIN[6+4*i_int],8) OR a_DataIN[5+4*i_int];
				a_rDataOut[i_int] := TO_REAL(di_Data) * r_scale + r_offset;
				ton_error.IN := FALSE;
			END_FOR
			b_next := TRUE;
			i_cycleCount := 0;
			r_out1 := a_rDataOut[1];
			r_out2 := a_rDataOut[2];
			r_out3 := a_rDataOut[3];
			r_out4 := a_rDataOut[4];
		ELSE
				i_cycleCount:= i_cycleCount + 1;
		END_IF
END_IF

IF  i_cycleCount = i_MaxRetries THEN
	i_RetryCount := i_retryCount + 1;
	b_next	:= TRUE;
	i_cycleCount := 0;	
ELSE
	b_error := FALSE;
END_IF

ton_error(IN := i_RetryCount = 3);
b_error := ton_error.Q;
END_METHOD

METHOD PRIVATE WriteReadRequest : BOOL
VAR_INPUT
	fastmode			: BOOL;
END_VAR

VAR_IN_OUT
	get				: ST_Wago750495_Get;
	b_enable		: BOOL;
END_VAR
VAR_INST
	b_next		        : BOOL;
	by_index			: BYTE;
	r_dummy				: REAL;
	st_EmptyData		: ST_Wago750495_Data;
	ftrig				: f_trig;
   	ProfilerActive     		: PROFILER;
	ProfilerReactive    	: PROFILER;
	by_StartIndex			 : BYTE;
	
	b_statusOK			: BOOL;
	i : INT;
	freq: REAL;
	Q_Old : REAL;
	P_Old : REAL;
	voltage : REAL;
	InverseFactor		: INT;
	ton_Release 		: ton := (PT := T#2s);
END_VAR
a_DataOUT[1].0 := set.b_EnableRegisterComm;
a_DataOUT[2] := set.e_statusQuery;
 

IF b_Enable THEN
	CASE by_Index OF
		0: 
			WriteIOCall(
				ID1_RQ := eWago750495_ACDataID.ActivePowerL1, 
				ID2_RQ := eWago750495_ACDataID.ActivePowerL2,
				ID3_RQ := eWago750495_ACDataID.ActivePowerL3,
				ID4_RQ := 0,
				COL_RQ := eWago750495_MeasureGroupID.ac,
				r_scale := 0.00001*InverseFactor,
				r_Offset := 0,
				b_next=>  b_next,
				r_out1 := get.Data.ar_ActivePower[1],
				r_out2 := get.Data.ar_ActivePower[2],
				r_out3 := get.Data.ar_ActivePower[3],
				r_out4 := r_dummy,
			);
			get.Data.ar_ActivePower[0] := get.Data.ar_ActivePower[1] + get.Data.ar_ActivePower[2] + get.Data.ar_ActivePower[3];
		1: 
			WriteIOCall(
				ID1_RQ := eWago750495_ACDataID.ReactivePowerL1,
				ID2_RQ := eWago750495_ACDataID.ReactivePowerL2,
				ID3_RQ := eWago750495_ACDataID.ReactivePowerL3,
				ID4_RQ := 0,
				COL_RQ := eWago750495_MeasureGroupID.ac,
				r_scale := 0.00001*InverseFactor,
				r_Offset := 0,
				b_next=>  b_next,
				r_out1 := get.Data.ar_ReactivePower[1],
				r_out2 := get.Data.ar_ReactivePower[2],
				r_out3 := get.Data.ar_ReactivePower[3],
				r_out4 := r_dummy,
			);
			get.Data.ar_ReactivePower[0] := get.Data.ar_ReactivePower[1] + get.Data.ar_ReactivePower[2] + get.Data.ar_ReactivePower[3];
		2: 
			WriteIOCall(
				ID1_RQ := eWago750495_ACDataID.VoltageL1N_RMS, 
				ID2_RQ := eWago750495_ACDataID.VoltageL2N_RMS,
				ID3_RQ := eWago750495_ACDataID.VoltageL3N_RMS,
				ID4_RQ := 0,
				COL_RQ := eWago750495_MeasureGroupID.ac,
				r_scale := 0.01,
				r_Offset := 0,
				b_next=>  b_next,
				r_out1 := get.Data.ar_VoltageLN[1],
				r_out2 := get.Data.ar_VoltageLN[2],
				r_out3 := get.Data.ar_VoltageLN[3],
				r_out4 := r_dummy,
			);
			get.data.ar_VoltageLN[0] := (get.Data.ar_VoltageLN[1] + get.Data.ar_VoltageLN[2] + get.Data.ar_VoltageLN[3]) / 3;
		3:
			WriteIOCall(
				ID1_RQ := eWago750495_ACDataID.VoltageL1L2_RMS, 
				ID2_RQ := eWago750495_ACDataID.VoltageL2L3_RMS,
				ID3_RQ := eWago750495_ACDataID.VoltageL3L1_RMS,
				ID4_RQ := 0,
				COL_RQ := eWago750495_MeasureGroupID.ac,
				r_scale := 0.01,
				r_Offset := 0,
				b_next=>  b_next,
				r_out1 := get.Data.ar_VoltageLL[1],
				r_out2 := get.Data.ar_VoltageLL[2],
				r_out3 := get.Data.ar_VoltageLL[3],
				r_out4 := r_dummy,
			);
			get.data.ar_VoltageLL[0] := (get.Data.ar_VoltageLL[1] + get.Data.ar_VoltageLL[2] + get.Data.ar_VoltageLL[3]) / 3;
		4: 
			WriteIOCall(
				ID1_RQ := eWago750495_ACDataID.CurrentL1_RMS, 
				ID2_RQ := eWago750495_ACDataID.CurrentL2_RMS,
				ID3_RQ := eWago750495_ACDataID.CurrentL3_RMS,
				ID4_RQ := eWago750495_ACDataID.CurrentN_RMS,
				COL_RQ := eWago750495_MeasureGroupID.ac,
				r_scale := 0.0001,
				r_Offset := 0,
				b_next=>  b_next,
				r_out1 := get.Data.ar_CurrentRMS[1],
				r_out2 := get.Data.ar_CurrentRMS[2],
				r_out3 := get.Data.ar_CurrentRMS[3],
				r_out4 := get.Data.ar_CurrentRMS[4],
			);
			get.Data.ar_CurrentRMS[0] := (get.Data.ar_CurrentRMS[1] + get.Data.ar_CurrentRMS[2] + get.Data.ar_CurrentRMS[3]) / 3;

		
		5: 
			WriteIOCall(
				ID1_RQ := eWago750495_ACDataID.FrequencyL1, 
				ID2_RQ := eWago750495_ACDataID.FrequencyL2,
				ID3_RQ := eWago750495_ACDataID.FrequencyL3,
				ID4_RQ := 0,
				COL_RQ := eWago750495_MeasureGroupID.ac,
				r_scale := 0.001,
				r_Offset := 0,
				b_next	=>  b_next,
				r_out1 := get.Data.ar_Frequency[1],
				r_out2 := get.Data.ar_Frequency[2],
				r_out3 := get.Data.ar_Frequency[3],
				r_out4 := r_dummy
			);
			get.Data.ar_Frequency[0] := (get.Data.ar_Frequency[1] + get.Data.ar_Frequency[2] + get.Data.ar_Frequency[3]) / 3;
		6: 
			WriteIOCall(
				ID1_RQ := eWago750495_ACDataID.PowerFactorL1, 
				ID2_RQ := eWago750495_ACDataID.PowerFactorL2,
				ID3_RQ := eWago750495_ACDataID.PowerFactorL3,
				ID4_RQ := 0,
				COL_RQ := eWago750495_MeasureGroupID.ac,
				r_scale := 0.01,
				r_Offset := 0,
				b_next=>  b_next,
				r_out1 := get.Data.ar_PowerFactor[1],
				r_out2 := get.Data.ar_PowerFactor[2],
				r_out3 := get.Data.ar_PowerFactor[3],
				r_out4 := r_dummy
			);	
			get.Data.ar_PowerFactor[0] := (get.Data.ar_PowerFactor[1] + get.Data.ar_PowerFactor[2] + get.Data.ar_PowerFactor[3]) / 3;
		7: 
			WriteIOCall(
				ID1_RQ := eWago750495_ACDataID.PhaseAngleL1, 
				ID2_RQ := eWago750495_ACDataID.PhaseAngleL2,
				ID3_RQ := eWago750495_ACDataID.PhaseAngleL3,
				ID4_RQ := 0,
				COL_RQ := eWago750495_MeasureGroupID.ac,
				r_scale := 0.01,
				r_Offset := 0,
				b_next=>  b_next,
				r_out1 := get.Data.ar_PhaseAngle[1],
				r_out2 := get.Data.ar_PhaseAngle[2],
				r_out3 := get.Data.ar_PhaseAngle[3],
				r_out4 := r_dummy
			);
			get.Data.ar_PhaseAngle[0] := (get.Data.ar_PhaseAngle[1] + get.Data.ar_PhaseAngle[2] +get.Data.ar_PhaseAngle[3]) / 3;
		8:
			WriteIOCall(
				ID1_RQ := eWago750495_ACDataID.ActiveEnergyExport, 
				ID2_RQ := eWago750495_ACDataID.ActiveEnergyImport,
				ID3_RQ := eWago750495_ACDataID.ActiveEnergyTotal,
				ID4_RQ := eWago750495_ACDataID.ReactiveEnergyTotal,
				COL_RQ := eWago750495_MeasureGroupID.ac,
				r_scale := 0.1,
				r_Offset := 0,
				b_next=>  b_next,
				r_out1 := get.Data.r_ActiveEnergyExport,
				r_out2 := get.Data.r_ActiveEnergyImport,
				r_out3 := get.Data.r_ActiveEnergyTotal,
				r_out4 := get.Data.r_ReactiveEnergyTotal
			);
			
			9:
			WriteIOCall(
				ID1_RQ := eWago750495_ACDataID.ActivePowerL1, 
				ID2_RQ := eWago750495_ACDataID.ReactivePowerL1,
				ID3_RQ := eWago750495_ACDataID.VoltageL1N_RMS,
				ID4_RQ := eWago750495_ACDataID.FrequencyL1,
				COL_RQ := eWago750495_MeasureGroupID.ac,
				r_scale := 0.00001 * inverseFactor,
				r_Offset := 0,
				b_next=>  b_next,
				r_out1 := get.Data.ar_ActivePower[1],
				r_out2 := get.Data.ar_ReactivePower[1],
				r_out3 := voltage,
				r_out4 := freq
			);
			10:
			WriteIOCall(
				ID1_RQ := eWago750495_ACDataID.ActivePowerL2, 
				ID2_RQ := eWago750495_ACDataID.ReactivePowerL2,
				ID3_RQ := eWago750495_ACDataID.ActivePowerL3,
				ID4_RQ := eWago750495_ACDataID.ReactivePowerL3,
				COL_RQ := eWago750495_MeasureGroupID.ac,
				r_scale := 0.00001 * inverseFactor,
				r_Offset := 0,
				b_next=>  b_next,
				r_out1 := get.Data.ar_ActivePower[2],
				r_out2 := get.Data.ar_ReactivePower[2],
				r_out3 := get.Data.ar_ActivePower[3],  
				r_out4 := get.Data.ar_ReactivePower[3],
			);
	END_CASE
END_IF

IF b_next THEN
	by_index := by_index + 1;
END_IF

by_StartIndex := SEL(fastmode, 0, 9);


ProfilerActive(START := get.Data.ar_ActivePower[2] = P_old);
ProfilerReactive(START := get.Data.ar_ReactivePower[1] = Q_old);

IF by_index = (9 + SEL(fastmode, -1, 2)) THEN
	by_index := by_StartIndex;
END_IF



InverseFactor := SEL(CTinverse, 1, -1);


b_statusOK := NOT (get.statusword.b_Error_L1 OR get.statusword.b_Error_L2 OR get.statusword.b_Error_L3);
ton_Release(IN := b_Enable AND b_statusOK);
IF ton_Release.Q AND fastmode THEN
	get.Data.ar_ReactivePower[0] := get.Data.ar_ReactivePower[1] + get.Data.ar_ReactivePower[2] + get.Data.ar_ReactivePower[3];
	get.Data.ar_ActivePower[0] := get.Data.ar_ActivePower[1] + get.Data.ar_ActivePower[2] + get.Data.ar_ActivePower[3];
	get.Data.ar_VoltageLN[0] := ABS(voltage) * 1000;
	get.Data.ar_Frequency[0] := ABS(freq) * 100;
		
	FOR i := 0 TO 4 DO
		get.Data.ar_ApparentPower[i] := SQRT(MAX(0, EXPT(get.Data.ar_ReactivePower[i], 2) + EXPT(get.Data.ar_ActivePower[i], 2)));
		get.Data.ar_CurrentRMS[i] := (get.Data.ar_ApparentPower[i] * 1000) / (MAX(1, get.Data.ar_VoltageLN[0]));
	END_FOR
	get.Data.ar_CurrentRMS[0] := (get.Data.ar_ApparentPower[0] * 1000) / (MAX(1, get.Data.ar_VoltageLN[0]) * 3);
	get.Data.ar_VoltageLL[0] := get.Data.ar_VoltageLN[0] * 1.73;
END_IF

ftrig(CLK:= FASTMODE XOR NOT b_statusOK);
IF ftrig.Q THEN
	get.Data := st_EmptyData;
END_IF

Q_Old := get.Data.ar_ReactivePower[1];
P_Old := get.Data.ar_ActivePower[2];
END_METHOD

END_FUNCTION_BLOCK

// ---- POUs/Functions-FBs-Programs/IO_modules/Beckhoff/FB_EK1100.TcPOU
FUNCTION_BLOCK FB_EK1100
VAR_OUTPUT
	state						AT %I* : UINT;
END_VAR

END_FUNCTION_BLOCK

// ---- POUs/Functions-FBs-Programs/IO_modules/Beckhoff/FB_EL3453.TcPOU
FUNCTION_BLOCK FB_EL3453

VAR_OUTPUT
	
	li_TimeVoltZeroCrossup	: ULINT;		
	PhaseStatus				 : ARRAY [1..3] OF ST_EL34xx_PhaseStatus;
	TotalStatus				 : ST_EL34xx_TotalStatus;
	r_PhaseVoltage			 : ARRAY [0..3] OF REAL;
	r_LineVoltage			 : ARRAY [0..3] OF REAL;
	r_Current				 : ARRAY [0..4] OF REAL;
	r_ActivePower			 : ARRAY [0..3] OF REAL;
	r_ReactivePower			 : ARRAY [0..3] OF REAL;
	r_ApparentPower			 : ARRAY [0..3] OF REAL;
	r_PowerFactor			 : ARRAY [0..3] OF REAL;
	r_Frequency				 : ARRAY [0..3] OF REAL;
	r_ActiveEnergy					: REAL;
	r_ActiveEnergyConsumed			: REAL;
	r_ActiveEnergySupplied			: REAL;
	r_VoltageUnbalance			  	: REAL;
	r_CurrentUnbalance				: REAL;
	r_ROCOF							: REAL;
	r_VoltageTHD					: ARRAY[0..3] OF REAL;
	r_CurrentTHD					: ARRAY[0..3] OF REAL;
	ui_EL3443BoxState		 AT %I*	: UINT;
END_VAR

VAR
	ReactiveDirection			: SINT;
	EL3453 : MDP5001_341_C93E75BD;
END_VAR

VAR_INPUT
	VoltageRatio			: REAL := 1;
	CurrentRatio			: INT := 200;
	CTInverse				: BOOL ; 
END_VAR

//current
r_Current[1]:= ValueConversion(DataSelector._C, ABS(EL3453.MDP5001_341_Input.MDP5001_341_L1_Classic_Current));
r_Current[2]:= ValueConversion(DataSelector._C, ABS(EL3453.MDP5001_341_Input.MDP5001_341_L2_Classic_Current));
r_Current[3]:= ValueConversion(DataSelector._C, ABS(EL3453.MDP5001_341_Input.MDP5001_341_L3_Classic_Current));
r_Current[0] := (r_Current[1] + r_Current[2] + r_Current[3]) / 3;

//voltage
r_PhaseVoltage[1] := ValueConversion(DataSelector._V, EL3453.MDP5001_341_Input.MDP5001_341_L1_Classic_Voltage);
r_PhaseVoltage[2] := ValueConversion(DataSelector._V, EL3453.MDP5001_341_Input.MDP5001_341_L2_Classic_Voltage);
r_PhaseVoltage[3] := ValueConversion(DataSelector._V, EL3453.MDP5001_341_Input.MDP5001_341_L3_Classic_Voltage);
r_PhaseVoltage[0] := (r_PhaseVoltage[1] + r_PhaseVoltage[2] + r_PhaseVoltage[3]) / 3;

r_LineVoltage[1]:= r_PhaseVoltage[1]* 1.73;
r_LineVoltage[2]:= r_PhaseVoltage[2]* 1.73;
r_LineVoltage[3]:= r_PhaseVoltage[3]* 1.73;
r_LineVoltage[0] := r_PhaseVoltage[0] * 1.73;

//active power
r_ActivePower[1]:= ValueConversion(DataSelector._P, EL3453.MDP5001_341_Input.MDP5001_341_L1_Classic_Active_power);
r_ActivePower[2]:= ValueConversion(DataSelector._P, EL3453.MDP5001_341_Input.MDP5001_341_L2_Classic_Active_power);
r_ActivePower[3]:= ValueConversion(DataSelector._P, EL3453.MDP5001_341_Input.MDP5001_341_L3_Classic_Active_power);
r_ActivePower[0] := (r_ActivePower[1] + r_ActivePower[2] + r_ActivePower[3]);


//Reactive power
IF EL3453.MDP5001_341_Input.MDP5001_341_Total_Reactive_Fundamental_Reactive_Power_Fund < 0 THEN ReactiveDirection := -1; ELSE ReactiveDirection := 1; END_IF
r_ReactivePower[1]:= ReactiveDirection * ValueConversion(DataSelector._Q, EL3453.MDP5001_341_Input.MDP5001_341_L1_Classic_Reactive_power);
r_ReactivePower[2]:= ReactiveDirection * ValueConversion(DataSelector._Q, EL3453.MDP5001_341_Input.MDP5001_341_L2_Classic_Reactive_power);
r_ReactivePower[3]:= ReactiveDirection * ValueConversion(DataSelector._Q, EL3453.MDP5001_341_Input.MDP5001_341_L3_Classic_Reactive_power);
r_ReactivePower[0] := EL3453.MDP5001_341_Input.MDP5001_341_Total_Reactive_Fundamental_Reactive_Power_Fund * CurrentRatio / 1000 * VoltageRatio * SEL(CTInverse, 1, -1);

//Apparent power
r_ApparentPower[1]:= ValueConversion(DataSelector._S, EL3453.MDP5001_341_Input.MDP5001_341_L1_Classic_Apparent_power);
r_ApparentPower[2]:= ValueConversion(DataSelector._S, EL3453.MDP5001_341_Input.MDP5001_341_L2_Classic_Apparent_power);
r_ApparentPower[3]:= ValueConversion(DataSelector._S, EL3453.MDP5001_341_Input.MDP5001_341_L3_Classic_Apparent_power);
r_ApparentPower[0] := (r_ApparentPower[1] + r_ApparentPower[2] + r_ApparentPower[3]);

//Active Energy
r_ActiveEnergy := ValueConversion(DataSelector._S, EL3453.MDP5001_341_Input.MDP5001_341_Total_Active_Fundamental_Active_Energy_Fund);
r_ActiveEnergySupplied := ValueConversion(DataSelector._S, EL3453.MDP5001_341_Input.MDP5001_341_Total_Active_Fundamental_Active_Negative_Energy_Fund);
r_ActiveEnergyConsumed := ValueConversion(DataSelector._S, EL3453.MDP5001_341_Input.MDP5001_341_Total_Active_Fundamental_Active_Positive_Energy_Fund);

//VoltageTHD
r_VoltageTHD[1] := EL3453.MDP5001_341_Input.MDP5001_341_L1_Advanced_Voltage_Total_Harmonic_Distortion;
r_VoltageTHD[2] := EL3453.MDP5001_341_Input.MDP5001_341_L2_Advanced_Voltage_Total_Harmonic_Distortion;
r_VoltageTHD[3] := EL3453.MDP5001_341_Input.MDP5001_341_L3_Advanced_Voltage_Total_Harmonic_Distortion;
r_VoltageTHD[0]	:= (r_VoltageTHD[1] + r_VoltageTHD[2] + r_VoltageTHD[3]) / 3;

//CurrentTHD
r_CurrentTHD[1] := EL3453.MDP5001_341_Input.MDP5001_341_L1_Advanced_Current_Total_Harmonic_Distortion;
r_CurrentTHD[2] := EL3453.MDP5001_341_Input.MDP5001_341_L2_Advanced_Current_Total_Harmonic_Distortion;
r_CurrentTHD[3] := EL3453.MDP5001_341_Input.MDP5001_341_L3_Advanced_Current_Total_Harmonic_Distortion;
r_CurrentTHD[0]	:= (r_CurrentTHD[1] + r_CurrentTHD[2] + r_CurrentTHD[3]) / 3;

//Frequecny
r_Frequency[1] := ValueConversion(DataSelector._F, EL3453.MDP5001_341_Input.MDP5001_341_L1_Classic_Frequency);
r_Frequency[2] := ValueConversion(DataSelector._F, EL3453.MDP5001_341_Input.MDP5001_341_L2_Classic_Frequency);
r_Frequency[3] := ValueConversion(DataSelector._F, EL3453.MDP5001_341_Input.MDP5001_341_L3_Classic_Frequency);
r_Frequency[0]	:= (r_Frequency[1] + r_Frequency[2] + r_Frequency[3]) / 3;


IF EL3453.MDP5001_341_Input.MDP5001_341_L1_Status_Voltage_Sign_Bit THEN
	li_TimeVoltZeroCrossup := EL3453.MDP5001_341_Input.MDP5001_341_L1_Timing_Voltage_Last_Zero_Crossing;
END_IF

r_PowerFactor [1] := Powerfactor(r_ActivePower[1], r_ApparentPower[1], r_ReactivePower[1]);
r_PowerFactor [2] := Powerfactor(r_ActivePower[2], r_ApparentPower[2], r_ReactivePower[2]);
r_PowerFactor [3] := Powerfactor(r_ActivePower[3], r_ApparentPower[3], r_ReactivePower[3]);
r_PowerFactor [0] := Powerfactor(r_ActivePower[0], r_ApparentPower[0], r_ReactivePower[0]);
r_VoltageUnbalance := LineUnbalance(r_LineVoltage[1], r_LineVoltage[2],r_LineVoltage[3]);
r_CurrentUnbalance := LineUnbalance(r_Current[1], r_Current[2], r_Current[3]);

TotalStatus.bit_GridDirection :=  EL3453.MDP5001_341_Input.MDP5001_341_Total_Status_Grid_Direction;
TotalStatus.bit_SystemState :=  EL3453.MDP5001_341_Input.MDP5001_341_Total_Status_System_State;

METHOD ValueConversion : REAL
VAR_INPUT
	selector		: DataSelector;
	IN				: LINT;
END_VAR

VAR
	totalRatio		: REAL;
	scale			: REAL;
END_VAR
scale := 0.001; //default

CASE selector OF
 	DataSelector._C:
		totalRatio := CurrentRatio;
	DataSelector._V:
		totalRatio := VoltageRatio;
	DataSelector._P, DataSelector._Q:
		totalRatio := CurrentRatio * VoltageRatio * SEL(CTInverse, 1, -1) / 1000;
	DataSelector._S, DataSelector._E:
		totalRatio := CurrentRatio * VoltageRatio / 1000;
	DataSelector._F:
		totalRatio := 1;
END_CASE

ValueConversion := TO_REAL(IN) * scale * totalRatio;
END_METHOD

END_FUNCTION_BLOCK

// ---- POUs/Objects/GenComm/FB_GenComm.TcPOU
FUNCTION_BLOCK FB_GenComm
VAR_INPUT
	Set				:	ST_Genset_Set;
END_VAR
VAR_OUTPUT
	Get				:	ST_Genset_Get;
END_VAR
VAR
	GenCommEnable		:	BOOL 	:= TRUE;
	OverwriteSetStruct	: 	BOOL 	:= FALSE;
	AGC150 				: 	FB_AGC150;
END_VAR

VAR_IN_OUT CONSTANT
	st_params 			: ST_GenComm_params;
END_VAR

AGC150(get := get, enable := GenCommEnable AND set.enable);

IF NOT OverwriteSetStruct THEN
	CASE st_params.GenControlProtocol OF
		eGenControlProtocol.AGC150:
			AGC150.set.ip := st_params.IP;
			AGC150.set.AutoStartStop := set.StartStop;
			AGC150.set.DroopEnable := FALSE;
			//defaults:
			AGC150.set.VoltRegulator := 0;
			AGC150.set.FreqRegulator := 0;
			AGC150.set.Pset := 0;
			AGC150.set.Qset := 0;
			AGC150.set.PFset := 1;	
			CASE set.GensetMode OF
				eGensetMode.Droop:
					AGC150.set.DroopEnable := TRUE;
					//AGC150.set.MainBreakerON := eOnOffState.Disable;
					AGC150.set.U_FDroopSet := set.U_FDroopSet;
					AGC150.set.VoltRegulator := set.Uset;
					AGC150.set.FreqRegulator := set.Fset;
					AGC150.set.bIslandModeEnable := TRUE; 
					AGC150.set.bFixedPowerEnable := FALSE;
				eGensetMode.Isochronous:
					AGC150.set.DroopEnable := FALSE;
					//AGC150.set.MainBreakerON := eOnOffState.Disable;
					AGC150.set.VoltRegulator := set.Uset;
					AGC150.set.FreqRegulator := set.Fset;
					AGC150.set.bIslandModeEnable := TRUE; 
					AGC150.set.bFixedPowerEnable := FALSE;
				eGensetMode.FixedPower:
					AGC150.set.bIslandModeEnable := FALSE; 
					AGC150.set.bFixedPowerEnable := TRUE;
					AGC150.set.DroopEnable := FALSE;
					//AGC150.set.MainBreakerON := eOnOffState.enable;
					AGC150.set.Pset := set.Pset;
					AGC150.set.Qset := set.Qset;
					AGC150.set.PFset := set.PFset;
			END_CASE
	END_CASE
END_IF

METHOD GetDiagnostics
VAR_IN_OUT
	AddError		: ARRAY [*] OF FB_AddErrorST;
	a_ActiveEvents	: ARRAY [*] OF ST_ErrorStruct;
	w_Index			: WORD;
END_VAR
	(*Comm error*)		AddError[w_Index](
					b_ErrorTrig				:= NOT get.CommunicationOK AND set.enable AND st_params.GenControlProtocol <> 0,
					out_ST_Error			:= a_ActiveEvents[w_Index],
					w_ErrorID				:= 1,
					e_ObjectID				:= eObject_ID.Genset,
					s_Message				:= 'communication not ok',
					e_sev					:= eSeverity.Info
				);
				w_Index := w_Index +1;
	
		(*Fuel low*)		AddError[w_Index](
					b_ErrorTrig				:= get.FuelLow OR get.FuelCritical,
					out_ST_Error			:= a_ActiveEvents[w_Index],
					w_ErrorID				:= 2,
					e_ObjectID				:= eObject_ID.Genset,
					s_Message				:= SEL(get.FuelCritical,'fuel at low level','fuel at critically low level'),
					e_sev					:= eSeverity.Info
				);
				w_Index := w_Index +1;
END_METHOD

END_FUNCTION_BLOCK

// ---- POUs/Objects/GenComm/FB_AGC150.TcPOU
FUNCTION_BLOCK FB_AGC150

VAR_IN_OUT
	get				: ST_GENSET_Get;
END_VAR

VAR_INPUT
	enable 	: BOOL;
	set 	: ST_AGC150_set;
END_VAR

VAR
	b_changeEndianess	:	BOOL	:=	FALSE;
	ComOKRelease		:   TON := (PT:= T#5S);
	MBWriteCoils		:	FB_MBWriteCoils;	// function 15
	CoilData			:	ARRAY[0..10] OF BYTE;
	StartCoilWrite		:	BOOL;
	
	MBWriteHolding		:	FB_MBWriteRegs;		// function 16
	HoldingData			:	ARRAY[0..4] OF WORD;
	StartHoldingWrite	:	BOOL;
	
	MBReadInputregs		:	FB_MBReadInputRegs;	//function 4
	InputRegData		:	ARRAY[0..27] OF WORD;
	StartInputRegRead	:	BOOL;
	
	MBReadInputs		:	FB_MBReadInputs;	//function 2
	InputData			:	ARRAY[0..2] OF BYTE;
	StartInputRead		:	BOOL;
	
	TransmissionDone	:	F_trig;
	bError				: BOOL;
	
	CommStep	:	UINT	:=	0;
	
	tpModbusDelay		: TP := (PT:= T#500MS);
END_VAR

tpModbusDelay();

IF NOT enable THEN
	commstep:= 0;
ELSIF (enable AND commstep = 0) THEN
	commstep := 1;
END_IF

MBWriteCoils(
	sIPAddr := set.IP,
	nTCPPort := 502,
	nUnitID := 1,//16#FF;
	nMBAddr := 0,//w_MBStartAddress,
	nQuantity := 50,
	cbLength := SIZEOF(CoilData),
	pSrcAddr := ADR(CoilData),
	bExecute := StartCoilWrite	//	<- werkt dit niet gewoon?
);

MBWriteHolding(
	sIPAddr := set.IP,
	nTCPPort := 502,
	nUnitID := 1,//16#FF;
	cbLength := SIZEOF(HoldingData),
	pSrcAddr := ADR(HoldingData),
	bExecute := StartHoldingWrite	//	<- werkt dit niet gewoon?
);
	
MBReadInputregs(
	sIPAddr := set.IP,
	nTCPPort := 502,
	nUnitID := 1,//16#FF;
	nMBAddr := 501,//w_MBStartAddress,
	nQuantity := 18,
	cbLength := SIZEOF(InputRegData),
	pDestaddr := ADR(InputRegData),
	bExecute := StartInputRegRead	//	<- werkt dit niet gewoon?
);

MBReadInputs(
	sIPAddr := set.IP,
	nTCPPort := 502,
	nUnitID := 1,//16#FF;
	nMBAddr := 501,//w_MBStartAddress,
	nQuantity := 5,
	cbLength := SIZEOF(InputData),
	pDestaddr := ADR(InputData),
	bExecute := StartInputRead	//	<- werkt dit niet gewoon?
);


CASE CommStep OF
	1: //Start MBWriteCoils
		CoilData[0].0 := set.GenOn = eOnoffState.Enable;
		CoilData[0].3 := set.GenOn = eOnoffState.Disable;
		
		CoilData[0].1 := set.GenBreakerOn = eOnoffState.Enable;
		CoilData[0].2 := set.GenBreakerOn = eOnoffState.Disable;
		
		CoilData[1].6 := set.GenAutoSyncOn = eOnoffState.Enable;
		CoilData[1].7 := set.GenAutoSyncOn = eOnoffState.Disable;
		
		CoilData[2].0 := set.bIslandModeEnable;
		CoilData[2].1 := set.bAMFModeEnable;
		CoilData[2].2 := set.bPeakshavingEnable;	
		CoilData[2].3 := set.bFixedPowerEnable;	
		CoilData[2].4 := set.bMPE;
		
		CoilData[3].0 := set.MainBreakerON = eOnoffState.Enable;
		CoilData[3].1 := set.MainBreakerON = eOnoffState.Disable;
		CoilData[3].2 := set.AutoStartStop;
		CoilData[3].3 := set.OperationMode = eGenOperationMode.ManualMode;
		CoilData[3].4 := set.OperationMode = eGenOperationMode.SemiAuto;	
		CoilData[3].5 := set.OperationMode = eGenOperationMode.Auto;	
		CoilData[3].6 := set.OperationMode = eGenOperationMode.Test;
		
		CoilData[6].0 := set.DroopEnable;
				
		StartCoilWrite := TRUE;
		Commstep := 2;
		
	2: //Wait for MBWriteCoils to finish
		StartCoilWrite := FALSE;
		bError := FALSE;
		IF NOT MBWriteCoils.bBusy THEN
			tpModbusDelay.IN := TRUE;
			IF NOT tpModbusDelay.Q THEN
				tpModbusDelay.IN := FALSE;
				IF NOT MBWriteCoils.bError THEN	
					Commstep := 3;
				 	//processdata
				ELSE
					//WriteFailed
					bError := TRUE;
					Commstep := 3;
				END_IF
			END_IF
		END_IF
		
	3: //Start MBWriteHolding
	 	MBWriteHolding.nMBAddr := 0;
		MBWriteHolding.nQuantity := 5;
		HoldingData[0] 	:= wordEndian(LIMIT(0, REAL_TO_UINT(set.Pset),100));
		HoldingData[1] 	:= wordEndian(LIMIT(60, REAL_TO_UINT(set.PFset),100));
		HoldingData[2] 	:= wordEndian(LIMIT(-100, REAL_TO_INT(set.Qset),100));
		HoldingData[3] 	:= wordEndian(LIMIT(-100, REAL_TO_INT(set.FreqRegulator),100));
		HoldingData[4] 	:= wordEndian(LIMIT(-100, REAL_TO_INT(set.VoltRegulator),100));
	
		StartHoldingWrite := TRUE;
		Commstep := 4;
		
	4: //Wait for MBWriteHolding to finish
		StartHoldingWrite := FALSE;
		
		IF NOT MBWriteHolding.bBusy THEN
			tpModbusDelay.IN := TRUE;
			IF NOT tpModbusDelay.Q THEN
				tpModbusDelay.IN := FALSE;
				IF NOT MBWriteHolding.bError THEN	
					Commstep := 5;
				 	//processdata
				ELSE
					//WriteFailed
					bError := TRUE;
					Commstep := 5;
				END_IF
			END_IF
		END_IF
		
	5: //Start MBReadInputregs
		StartInputRegRead := TRUE;
		Commstep := 6;
		
	6: //Wait for MBReadInputregs to finish
		StartInputRegRead := FALSE;
		IF NOT MBReadInputregs.bBusy THEN
			tpModbusDelay.IN := TRUE;
			IF NOT tpModbusDelay.Q THEN
				tpModbusDelay.IN := FALSE;
				IF NOT MBReadInputregs.bError THEN		
					get.ar_Linevoltage[phases.L1]	:= WORD_TO_REAL(WordEndian(InputRegData[0]));
					get.ar_Linevoltage[phases.L2]	:= WORD_TO_REAL(WordEndian(InputRegData[1]));
					get.ar_Linevoltage[phases.L3]	:= WORD_TO_REAL(WordEndian(InputRegData[2]));
					get.ar_LineVoltage[phases.AVG]	:= (get.ar_Linevoltage[phases.L1]+ get.ar_Linevoltage[phases.L2] + get.ar_Linevoltage[phases.L3]) / 3;
					
					get.ar_Phasevoltage[phases.L1]	:= WORD_TO_REAL(wordendian(InputRegData[3]));
					get.ar_Phasevoltage[phases.L2]	:= WORD_TO_REAL(wordendian(InputRegData[4]));
					get.ar_Phasevoltage[phases.L3]	:= WORD_TO_REAL(wordendian(InputRegData[5]));
					get.ar_PhaseVoltage[phases.AVG]	:= (get.ar_Phasevoltage[phases.L1]+ get.ar_Phasevoltage[phases.L2] + get.ar_Phasevoltage[phases.L3]) / 3;
							 
					get.ar_Frequency[phases.L1]		:= WORD_TO_REAL(wordendian(InputRegData[6])) / 100;
					get.ar_Frequency[phases.L2]		:= WORD_TO_REAL(wordendian(InputRegData[7])) / 100;
					get.ar_Frequency[phases.L3]		:= WORD_TO_REAL(wordendian(InputRegData[8])) / 100;
					get.ar_Frequency[phases.AVG]		:= (get.ar_Frequency[phases.L1]+ get.ar_Frequency[phases.L2] + get.ar_Frequency[phases.L3]) / 3;
							 
					get.ar_Current[phases.L1]	:= WORD_TO_REAL(wordendian(InputRegData[12]));
					get.ar_Current[phases.L2]	:= WORD_TO_REAL(wordendian(InputRegData[13]));
					get.ar_Current[phases.L3]	:= WORD_TO_REAL(wordendian(InputRegData[14]));
					get.ar_Current[phases.AVG] := (get.ar_Current[phases.L1] + get.ar_Current[phases.L2]  + get.ar_Current[phases.L3]) / 3;
						   
					get.ar_ActivePower[phases.L1]	:= WORD_TO_REAL(wordendian(InputRegData[15]));
					get.ar_ActivePower[phases.L2]	:= WORD_TO_REAL(wordendian(InputRegData[16]));
					get.ar_ActivePower[phases.L3]	:= WORD_TO_REAL(wordendian(InputRegData[17]));
					get.ar_ActivePower[phases.AVG]	:= (get.ar_ActivePower[phases.L1] + get.ar_ActivePower[phases.L2]  + get.ar_ActivePower[phases.L3]);
					
					Get.ar_ApparentPower[phases.AVG] := (get.ar_Current[phases.L1] * get.ar_PhaseVoltage[1] + get.ar_Current[phases.L2] * get.ar_PhaseVoltage[2] + get.ar_Current[phases.L3] * get.ar_PhaseVoltage[3]) / 1000;
					Get.ar_ReactivePower[phases.AVG] := ReactivePower(Get.ar_ApparentPower[phases.AVG], get.ar_ActivePower[phases.AVG], 0);  
					Get.ar_PowerFactor[phases.AVG] := PowerFactor(get.ar_ActivePower[phases.AVG],Get.ar_ApparentPower[phases.AVG], Get.ar_ReactivePower[phases.AVG]);
					Commstep := 7;
				ELSE
					//WriteFailed
					bError := TRUE;
					Commstep := 7;
				END_IF
			END_IF
		END_IF		
		
	7: //Start MBReadInputs
		StartInputRead := TRUE;
		Commstep := 8;
		
	8: //Wait for MBReadInputs to finish
		StartInputRead := FALSE;
		IF NOT MBReadInputs.bBusy THEN
			tpModbusDelay.IN := TRUE;
			IF NOT tpModbusDelay.Q THEN
				tpModbusDelay.IN := FALSE;
				IF NOT MBReadInputs.bError THEN
					get.bGenBreakerClosed 	:= InputData[0].0;  
					
					get.bMainBreakerClosed 	:= InputData[0].1;
					get.bGenRunning 		:= InputData[0].3;
					get.bGenVoltFreqOK 		:= InputData[0].4;
					get.bMainsFailure 		:= InputData[0].5;
					
					IF InputData[0].6 THEN	get.eActiveGenMode := eGenOperationMode.BlockMode;
					ELSIF InputData[0].7 THEN	get.eActiveGenMode := eGenOperationMode.ManualMode;
					ELSIF InputData[1].0 THEN	get.eActiveGenMode := eGenOperationMode.SemiAuto;
					ELSIF InputData[1].1 THEN	get.eActiveGenMode := eGenOperationMode.Auto;
					ELSIF InputData[1].2 THEN	get.eActiveGenMode := eGenOperationMode.Test;
					END_IF
					
					get.bIslandModeActive := InputData[1].5;
					get.bMainsFailure	:=	InputData[1].6;
					get.bPeakshaveActive := InputData[1].7;
					get.bFixedPowerActive := InputData[2].0;				
					Commstep := 9;
				ELSE
					//WriteFailed
					bError := TRUE;
					Commstep := 9;
				END_IF
			END_IF
		END_IF

	9: //Start MBWriteHolding
		MBWriteHolding.nMBAddr := 4125;
		MBWriteHolding.nQuantity := 1;
		HoldingData[0] 	:= wordEndian(LIMIT(0, REAL_TO_UINT(set.U_Fdroopset * 10), 100));

		StartHoldingWrite := TRUE;
		Commstep := 10;
		
	10: //Wait for MBWriteHolding to finish
		StartHoldingWrite := FALSE;
		
		IF NOT MBWriteHolding.bBusy THEN
			tpModbusDelay.IN := TRUE;
			IF NOT tpModbusDelay.Q THEN
				tpModbusDelay.IN := FALSE;
				IF NOT MBWriteHolding.bError THEN	
					Commstep := 1;
				 	//processdata
				ELSE
					//WriteFailed
					bError := TRUE;
					Commstep := 1;
				END_IF
			END_IF
		END_IF
END_CASE

ComOKRelease(IN:= NOT bError AND Commstep <>0, Q => get.CommunicationOK);

METHOD WordEndian : WORD
VAR_INPUT
	IN		: WORD;
END_VAR
IF b_changeEndianess THEN
	WordEndian := HOST_TO_BE16(IN);
ELSE
	WordEndian := IN;
END_IF
END_METHOD

END_FUNCTION_BLOCK

// ---- POUs/MAIN_Slow.TcPOU
PROGRAM MAIN_Slow
VAR
	{ attribute 'TcHmiSymbol.Hide' }
	monitor								: REFERENCE TO ST_System_Monitor;
	control								: ST_system_Control;
	
	{ attribute 'TcHmiSymbol.Hide' }				
	b_validref							: BOOL;
	//InterMachineCom							: FB_InterMachineCommunication;
END_VAR

Errorhandling(b_ClearEvents := control.control.b_ClearHistory);
//Eventlog(stparams:=Settings.MachineParams.Eventlogger);
//InterMachineCom(monitor:=monitor);
//Get refs of monitoring from fast cycle
monitor REF= MAIN_fast.monitor;
monitor.controlfb REF= control;


b_validref := __ISVALIDREF(monitor.powerstack) AND 
		__ISVALIDREF(monitor.battery) AND 
		__ISVALIDREF(monitor.neutraltransformer) AND
		__ISVALIDREF(monitor.powermonitor) AND
		__ISVALIDREF(monitor.protections) AND
		__ISVALIDREF(monitor.ACswitchgear) AND
		__ISVALIDREF(monitor.AcDcCharger) AND
		__ISVALIDREF(monitor.internalpsu) AND
		__ISVALIDREF(monitor.peakshavebox); // AND __ISVALIDREF(monitor)

IF b_validref THEN
	ControlManager(
		Monitor:=monitor,
		operation := control.Operation,
		control := control.control);
		control.HardSettings := ControlManager.PLCpersistvars.Hardsettings;
		control.SoftSettings := ControlManager.PLCpersistvars.Softsettings;

//VERY IMPORTANT. This closes the initialization after the slow cycle is executed the first time.
GVL.b_initCycle := FALSE;
END_IF

END_PROGRAM

// ---- POUs/Datalogger/DataLogging/ArrayVariables.TcPOU
PROGRAM ArrayVariables
VAR_IN_OUT CONSTANT
	Monitoring			: ST_System_Monitor;
END_VAR



VAR
	HeaderArray			: ARRAY [1..Datalogger.NUMBEROFCOLUMNS] OF STRING;
	VariableArray		: ARRAY [1..Datalogger.NUMBEROFCOLUMNS] OF STRING;
	milliSec			: STRING;
END_VAR


//When Removing or Adding file always change 'WriteToFile.NUMBEROFCOLUMNS' to the amount of variables

HeaderArray[1]   :='Time';
HeaderArray[2]   :='ErrorID';			      								
HeaderArray[3]   :='Severity'; 		                        
HeaderArray[4]   :='Message'; 		                        
HeaderArray[5]   :='System state';
HeaderArray[6]   :='Powerstack state';   		                        
HeaderArray[7]   :='BMS state'; 			        
HeaderArray[8]   :='Cooling state';
//HeaderArray[9]   :='T CMchoke L2 core';  		        
//HeaderArray[10]   :='T CMchoke L3 Inner'; 			        
//HeaderArray[11]   :='T CMchoke L3 Outer';
//HeaderArray[12]   :='T CMchoke L3 core'; 		                        
//HeaderArray[13]  :='T CMchoke DC Inner';		        
//HeaderArray[14]  :='T CMchoke DC Outer';
//HeaderArray[15]   :='T CMchoke DC core';			        
//HeaderArray[16]  :='T GrChoke L1 Inner';              	        
//HeaderArray[17]  :='T GrChoke L1 Outer';
//HeaderArray[18]  :='T GrChoke L1 core';			        
//HeaderArray[19]  :='T GrChoke L2 Inner'; 			        
//HeaderArray[20]  :='T GrChoke L2 Outer';
//HeaderArray[21]  :='T GrChoke L2 core';					        
//HeaderArray[22]  :='T GrChoke L3 Inner';                      
//HeaderArray[23]  :='T GrChoke L3 Outer';
//HeaderArray[24]  :='T GrChoke L3 core';		                        
//HeaderArray[25]  :='T AC Caps bottom';                        
//HeaderArray[26]  :='T AC Caps top';                        
//HeaderArray[27]  :='T DC Caps';                        
//HeaderArray[28]  :='T Fancoil Compartment';                        
//HeaderArray[29]  :='T air inlet';              	        
//HeaderArray[30]  :='T air outlet (fancoil)';			        
//HeaderArray[31]  :='T Water inlet (fancoil)';                        
//HeaderArray[32]  :='T Water outlet (fancoil)';                        
//HeaderArray[33]  :='T DC busbar CM choke';	                        
//HeaderArray[34]  :='T AC busbar CM choke L3'; 
//HeaderArray[35]  :='T AC busbar Output L1';                        
//HeaderArray[36]  :='Active Power';	                        
//HeaderArray[37]  :='Total current';	                        
                     
																													                                                                                       
VariableArray[1]   :=  GVL.s_SystemTime;
VariableArray[2]   :=  TO_STRING(Monitoring.powerstack.PowermoduleMaster.AddTemperatures.r_ambient);
VariableArray[3]   :=  TO_STRING(Monitoring.powerstack.PowermoduleMaster.r_TemperatureInverter);
VariableArray[4]   :=  TO_STRING(Monitoring.powerstack.PowermoduleMaster.AddTemperatures.r_CMchokeInner[1]);
VariableArray[5]   :=  TO_STRING(Monitoring.powerstack.PowermoduleMaster.AddTemperatures.r_CMchokeOuter[1]);
VariableArray[6]   :=  TO_STRING(Monitoring.powerstack.PowermoduleMaster.r_TemperatureCMChoke[1]);
VariableArray[7]   :=  TO_STRING(Monitoring.powerstack.PowermoduleMaster.AddTemperatures.r_CMchokeInner[2]);
VariableArray[8]   :=  TO_STRING(Monitoring.powerstack.PowermoduleMaster.AddTemperatures.r_CMchokeOuter[2]);
VariableArray[9]   :=  TO_STRING(Monitoring.powerstack.PowermoduleMaster.r_TemperatureCMChoke[2]);
VariableArray[10]   :=  TO_STRING(Monitoring.powerstack.PowermoduleMaster.AddTemperatures.r_CMchokeInner[3]);
VariableArray[11]   :=  TO_STRING(Monitoring.powerstack.PowermoduleMaster.AddTemperatures.r_CMchokeOuter[3]);
VariableArray[12]   :=  TO_STRING(Monitoring.powerstack.PowermoduleMaster.r_TemperatureCMChoke[3]);
VariableArray[13]   :=  TO_STRING(Monitoring.powerstack.PowermoduleMaster.AddTemperatures.r_CMchokeInner[4]);
VariableArray[14]   :=  TO_STRING(Monitoring.powerstack.PowermoduleMaster.AddTemperatures.r_CMchokeOuter[4]);
VariableArray[15]   :=  TO_STRING(Monitoring.powerstack.PowermoduleMaster.r_TemperatureCMChoke[4]);
VariableArray[16]   :=  TO_STRING(Monitoring.powerstack.PowermoduleMaster.AddTemperatures.r_GrChokeInner[1]);
VariableArray[17]   :=  TO_STRING(Monitoring.powerstack.PowermoduleMaster.AddTemperatures.r_GrChokeOuter[1]);
VariableArray[18]   :=  TO_STRING(Monitoring.powerstack.PowermoduleMaster.r_TemperatureGridChoke[1]);
VariableArray[19]   :=  TO_STRING(Monitoring.powerstack.PowermoduleMaster.AddTemperatures.r_GrChokeInner[2]);
VariableArray[20]   :=  TO_STRING(Monitoring.powerstack.PowermoduleMaster.AddTemperatures.r_GrChokeOuter[2]);
VariableArray[21]   :=  TO_STRING(Monitoring.powerstack.PowermoduleMaster.r_TemperatureGridChoke[2]);
VariableArray[22]   :=  TO_STRING(Monitoring.powerstack.PowermoduleMaster.AddTemperatures.r_GrChokeInner[3]);
VariableArray[23]   :=  TO_STRING(Monitoring.powerstack.PowermoduleMaster.AddTemperatures.r_GrChokeOuter[3]);
VariableArray[24]   :=  TO_STRING(Monitoring.powerstack.PowermoduleMaster.r_TemperatureGridChoke[3]);
VariableArray[25]   :=  TO_STRING(Monitoring.powerstack.PowermoduleMaster.AddTemperatures.r_ACCapsBottom);
VariableArray[26]   :=  TO_STRING(Monitoring.powerstack.PowermoduleMaster.AddTemperatures.r_ACCapsTop);
VariableArray[27]   :=  TO_STRING(Monitoring.powerstack.PowermoduleMaster.AddTemperatures.r_DCCaps);
VariableArray[28]   :=  TO_STRING(Monitoring.powerstack.PowermoduleMaster.AddTemperatures.r_FancoilCompartement);
VariableArray[29]   :=  TO_STRING(Monitoring.powerstack.PowermoduleMaster.AddTemperatures.r_AirInletModule);
VariableArray[30]   :=  TO_STRING(Monitoring.powerstack.PowermoduleMaster.AddTemperatures.r_AirOutletFancoil);
VariableArray[31]   :=  TO_STRING(Monitoring.powerstack.PowermoduleMaster.AddTemperatures.r_WaterInletFancoil);
VariableArray[32]   :=  TO_STRING(Monitoring.powerstack.PowermoduleMaster.AddTemperatures.r_WaterOutletFancoil);
VariableArray[33]   :=  TO_STRING(Monitoring.powerstack.PowermoduleMaster.AddTemperatures.r_DCbusbarCMChoke);
VariableArray[34]   :=  TO_STRING(Monitoring.powerstack.PowermoduleMaster.AddTemperatures.r_ACbusbarCMchoke);
VariableArray[35]   :=  TO_STRING(Monitoring.powerstack.PowermoduleMaster.AddTemperatures.r_ACbusbarOutput);
VariableArray[36]   :=  TO_STRING(Monitoring.powerstack.PowermoduleMaster.PowerMonitor.r_ActivePower[0]);
VariableArray[37]   :=  TO_STRING(Monitoring.powerstack.PowermoduleMaster.PowerMonitor.r_Current[1]);

END_PROGRAM

// ---- POUs/Datalogger/DataLogging/Datalogger.TcPOU
PROGRAM Datalogger
VAR_IN_OUT CONSTANT
	monitoring			: ST_System_Monitor;
END_VAR

VAR
	FB_Datalogger					:FB_Datalogger;
END_VAR
VAR CONSTANT
	MAXLREALTOSTRINGLENGTH			: UDINT := 30;	
	NUMBEROFCOLUMNS					: UDINT := 40;													// Total number of columns
	TOTALNUMBEROFROWS				: UDINT := 86400;										    	// Total number of rows in one file (Depends of logtime)
	INCREOFROWS						: UDINT := 5;													// Amount of rows to write at once
	BUFFERMEM						: UDINT := 150;													// Effects file size
	NUMBEROFELEMENTS				: UDINT := NUMBEROFCOLUMNS * INCREOFROWS;						// > NUMBEROFCOLUMNS * INCREOFROWS
	MARGEDATAUSAGE					: REAL  := 0.05;												// 5% Standard marge (95% of storage gets used)
END_VAR
VAR PERSISTENT
	//Datalog presis 
	udi_MaxAmoutOfFiles									: UDINT;								// Max amount of files (30Mb = 12000 ROWS = 10min log)
	udi_AmountOfFiles									: UDINT;
	b_FileNotClosed										: BOOL;
	ui_FileNotClosed									: UINT; 
	a_LogFilesCreated									: ARRAY [0..10000] OF STRING(30);
END_VAR

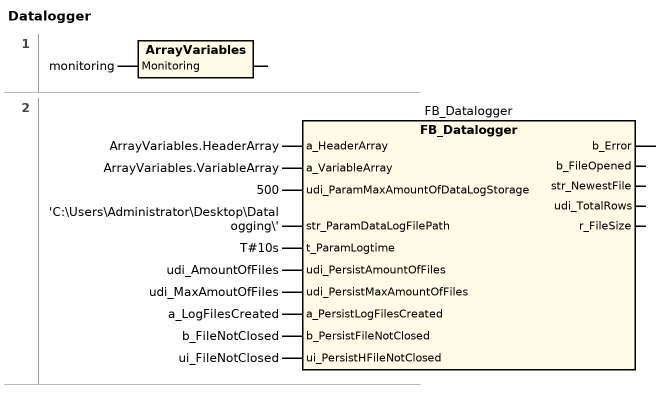
// NETWORK 1
ArrayVariables(Monitoring := monitoring);

// NETWORK 2
FB_Datalogger(
    a_HeaderArray := ArrayVariables.HeaderArray,
    a_VariableArray := ArrayVariables.VariableArray,
    udi_ParamMaxAmountOfDataLogStorage := 500,
    str_ParamDataLogFilePath := 'C:\Users\Administrator\Desktop\Datalogging\',
    t_ParamLogtime := T#10s,
    udi_PersistAmountOfFiles := udi_AmountOfFiles,
    udi_PersistMaxAmountOfFiles := udi_MaxAmoutOfFiles,
    a_PersistLogFilesCreated := a_LogFilesCreated,
    b_PersistFileNotClosed := b_FileNotClosed,
    ui_PersistHFileNotClosed := ui_FileNotClosed);

END_PROGRAM

// ---- POUs/Datalogger/FUNCTIONBLOCKS/FB_Datalogger.TcPOU
FUNCTION_BLOCK FB_Datalogger
VAR_IN_OUT
	Event			: ST_ErrorStruct;
END_VAR

VAR_IN_OUT CONSTANT
	Monitor			: ST_System_Monitor;
END_VAR

VAR_INPUT
	sTime								: STRING;
	sDate								: STRING;
	udi_ParamMaxAmountOfDataLogStorage	: UDINT;
	str_ParamDataLogFilePath			: STRING;
	t_ParamLogtime						: TIME;
END_VAR
VAR_OUTPUT
	b_Error							: BOOL := FALSE;
	b_FileOpened					: BOOL;
	str_NewestFile					: STRING;
	udi_TotalRows					: UDINT := 0;
	r_FileSize						: REAL; 
END_VAR
VAR_IN_OUT
	udi_PersistAmountOfFiles		: UDINT;
	udi_PersistMaxAmountOfFiles		: UDINT;
	a_PersistLogFilesCreated		: ARRAY [0..10000] OF STRING(30);
	b_PersistFileNotClosed			: BOOL;
	ui_PersistHFileNotClosed		: UINT;
END_VAR
VAR						
	//FB Open-Write-Close file
	fileOpen						: FB_FileOpen;
	fileWrite						: FB_FileWrite;
	fileClose						: FB_FileClose;
	fileCloseNotClosed				: FB_FileClose;

	//Buffer	
	FB_CsvBuffer					: FB_CSVWriter;
	bufferMemory					: ARRAY[1..Datalogger.BUFFERMEM] OF STRING;	
	cleardata						: ARRAY[1..Datalogger.BUFFERMEM] OF STRING; 
	
	//Data 
	DataVar							: ARRAY [1..Datalogger.NUMBEROFELEMENTS] OF STRING;
	filePath						: STRING:='C:\users\Administrator\desktop\datalogging\';				//Filepath, name gets created in prog
	filePathAmount					: STRING;
	
	//Header
	DataHeader						: ARRAY [1..Datalogger.NUMBEROFCOLUMNS] OF STRING;
	
	//Var
	ton_log							: TON;
	step							: INT := 0;
	cntr1							: UDINT := 1;
	idx								: UDINT := 1;
	elementcounter					: UDINT := 0;
	increment						: UDINT := 0;
	logdelay						: UDINT := 0;
	
	//Log data limit
	idx1								: UDINT;
	deleteFile							: FB_FileDelete;
	trig								: R_TRIG;
	Filesize							: FB_EnumFindFileEntry;
	b_Readsize							: BOOL;
END_VAR

//Data limiter **
//Limint amount of files
r_FileSize := (DWORD_TO_REAL(Filesize.stFindFile.fileSize.dwLowPart)/1022938);

//Files need to be fully completed (Standard = 15 files) 
IF udi_PersistAmountOfFiles < 1 THEN
	udi_PersistMaxAmountOfFiles := 15;
ELSIF udi_PersistAmountOfFiles >= 1  AND r_FileSize > 0 AND NOT b_PersistFileNotClosed THEN 
	udi_PersistMaxAmountOfFiles := REAL_TO_UDINT(udi_ParamMaxAmountOfDataLogStorage / (r_FileSize*(1+Datalogger.MARGEDATAUSAGE)));
END_IF


trig(CLK:=b_FileOpened , Q=> );

//Move data up the array
IF trig.Q THEN
	FOR idx1:= udi_PersistMaxAmountOfFiles TO 1 BY -1 DO
		a_PersistLogFilesCreated[idx1]:=a_PersistLogFilesCreated[idx1-1];
	END_FOR
a_PersistLogFilesCreated[0]:=str_NewestFile;
END_IF

//Delete oldest file
deleteFile(
	sNetId:= , 
	sPathName:= a_PersistLogFilesCreated[udi_PersistMaxAmountOfFiles], 
	ePath:= , 
	bExecute:= trig.Q, 
	tTimeout:=, 
	bBusy=> , 
	bError=> , 
	nErrId=> );

//Read file size
IF b_FileOpened AND udi_PersistAmountOfFiles > 1 THEN
	b_Readsize := TRUE;
ELSE 
	b_Readsize := FALSE;
END_IF
	
Filesize(
	sNetId:= , 
	sPathName:= a_PersistLogFilesCreated[1] , 
	eCmd:= , 
	bExecute:= b_Readsize, 
	tTimeout:= , 
	bBusy=> , 
	bError=> , 
	nErrID=> , 
	bEOE=> , 
	stFindFile=> );


	
//Data logger**
ton_log(IN:=NOT ton_log.Q , PT:=t_ParamLogtime , Q=> , ET=> );       


filePath := CONCAT(str_ParamDataLogFilePath, CONCAT(sTime , ' DataLogging.csv'));

//FB open - write - close
fileOpen(
	sNetId:= , 
	sPathName:=filePath , 
	nMode:=FOPEN_MODEWRITE OR FOPEN_MODETEXT , 
	ePath:=PATH_GENERIC , 
	tTimeout:=T#3S);

fileWrite(
	sNetId:= , 
	hFile:=fileOpen.hFile , 
	pWriteBuff:=ADR(bufferMemory) , 
	cbWriteLen:=SIZEOF(bufferMemory) , 
	tTimeout:=T#3S);	
		
fileClose(
	sNetId:= , 
	hFile:=fileOpen.hFile , 
	tTimeout:=T#3S);


 
//Start delay
IF 	ton_log.Q AND logdelay <= 2 THEN 
	logdelay := logdelay + 1;
END_IF


IF logdelay >= 2 THEN 
	
//Var loop
IF ton_log.Q AND NOT b_Error THEN
	FOR cntr1 := 1 TO Datalogger.NUMBEROFCOLUMNS DO
		DataVar[elementcounter + cntr1] := a_VariableArray[cntr1];
	END_FOR
	elementCounter := elementCounter + Datalogger.NUMBEROFCOLUMNS;
	udi_TotalRows := udi_TotalRows + 1;
END_IF	

	
CASE step OF

//Condition
0:		IF  NOT b_Error AND NOT b_FileOpened THEN
			step:= 10;
		ELSIF  udi_TotalRows >= Datalogger.INCREOFROWS * (increment+1) AND NOT b_Error AND b_FileOpened AND udi_TotalRows <= Datalogger.TOTALNUMBEROFROWS THEN
			step:= 30;
		ELSIF udi_TotalRows >= Datalogger.TOTALNUMBEROFROWS AND NOT b_Error THEN
			step:= 50;
		ELSIF NOT fileOpen.bError AND NOT fileWrite.bError AND NOT fileClose.bError THEN
			b_Error := FALSE;
		ELSE 
			step:= 0;
		END_IF


//Opening file - check if old file is closed (due random shutdown)
10:		fileOpen.bExecute:=TRUE;
	
		IF fileOpen.bBusy THEN
			fileOpen.bExecute:=FALSE;
			step:=11;
		END_IF

//Waiting for the file to be open
11: 	IF NOT fileOpen.bBusy AND NOT fileOpen.bError THEN
			b_FileOpened := TRUE;
			
			IF b_PersistFileNotClosed THEN
				fileCloseNotClosed.bExecute:= TRUE;
			END_IF
			//If file not closed due random shutdown 
			fileCloseNotClosed(
				sNetId:= , 
				hFile:=ui_PersistHFileNotClosed , 
				tTimeout:=T#3S);
			
			str_NewestFile := filePath;
			IF udi_PersistAmountOfFiles < udi_PersistMaxAmountOfFiles THEN
				udi_PersistAmountOfFiles:= udi_PersistAmountOfFiles+1;
				ui_PersistHFileNotClosed := fileopen.hFile;
				fileCloseNotClosed.bExecute:= FALSE;
				b_PersistFileNotClosed := TRUE;
			END_IF
			step:=20;
		ELSE
			b_Error:=TRUE;	
			step:=0;
		END_IF

//Load buffer with header
20:		FOR idx:=1 TO Datalogger.NUMBEROFCOLUMNS  DO
		
			IF idx=1 THEN
				FB_CsvBuffer.eCmd:=eEnumCmd_First;
			ELSE
				FB_CsvBuffer.eCmd:=eEnumCmd_Next;
			END_IF
            
			IF idx MOD Datalogger.NUMBEROFCOLUMNS=0 AND idx>1 THEN				
				FB_CsvBuffer.bLF:=TRUE;
			ELSE
				FB_CsvBuffer.bLF:=FALSE;
			END_IF
						
			FB_CsvBuffer.putValue:=STRING_TO_CSVFIELD(eventtype.Column[idx].s_header,bQm:=FALSE);
			
			
			FB_CsvBuffer(
				pBuffer		:= ADR(bufferMemory) , 
				cbBuffer	:= SIZEOF(bufferMemory) , 
				bOk=> , 
				cbSize=> , 
				cbFree=> , 
				nFields=> , 
				nRecords=> , 
				cbWrite=> );

		END_FOR
		step:=21;
		
//Write header
21:		fileWrite.bExecute:=TRUE;
	
		IF fileWrite.bBusy THEN
			fileWrite.bExecute:=FALSE;
			step:=22;
		END_IF
		
22: 	IF NOT fileWrite.bBusy AND NOT fileWrite.bError  THEN
			step:=0;
			bufferMemory:=cleardata;
		ELSE  
			b_Error:=TRUE;
			step:=0;
		END_IF

//Load buffer with data variables
30:		FOR idx:=1 TO Datalogger.NUMBEROFCOLUMNS * Datalogger.INCREOFROWS  DO
		
			IF idx=1 THEN
				FB_CsvBuffer.eCmd:=eEnumCmd_First;
			ELSE
				FB_CsvBuffer.eCmd:=eEnumCmd_Next;
			END_IF
            
			IF idx MOD Datalogger.NUMBEROFCOLUMNS=0 AND idx>1 THEN				
				FB_CsvBuffer.bLF:=TRUE;
			ELSE
				FB_CsvBuffer.bLF:=FALSE;
			END_IF
						
			FB_CsvBuffer.putValue:=STRING_TO_CSVFIELD(DataVar[idx],bQm:=FALSE);
			
			
			FB_CsvBuffer(
				pBuffer		:= ADR(bufferMemory) , 
				cbBuffer	:= SIZEOF(bufferMemory) , 
				bOk=> , 
				cbSize=> , 
				cbFree=> , 
				nFields=> , 
				nRecords=> , 
				cbWrite=> );

		END_FOR
		step:=31;

//Write var data 
31: 	fileWrite.bExecute:=TRUE;
	
		IF fileWrite.bBusy THEN
			fileWrite.bExecute:=FALSE;
			elementCounter := 0;
			step:=32;
		END_IF
		
32: 	IF NOT fileWrite.bBusy AND NOT fileWrite.bError THEN
			step:=40;
			bufferMemory:=cleardata;
		ELSE  
			b_Error:=TRUE;
			step:=0;
		END_IF
	
//Totalrows = TOTALNUMBEROFROWS
40: 	IF udi_TotalRows < Datalogger.TOTALNUMBEROFROWS THEN
			increment := increment + 1;
			step:=0;
		ELSE
			step:=50;
		END_IF
	
//Closing the file
50: 	fileClose.bExecute:=TRUE;
		
		IF fileClose.bBusy THEN
			fileClose.bExecute:=FALSE;
			b_PersistFileNotClosed:= FALSE;
			step:=51;
		END_IF

//Waiting for the file to be closed
51: IF NOT fileClose.bBusy AND NOT fileClose.bError THEN
			b_FileOpened:= FALSE;
			increment:= 0;
			udi_TotalRows:= 0;
			step:=0;
		ELSE
			b_Error:= TRUE;
			step:=0;
		END_IF

END_CASE

END_IF

METHOD EventType : BOOL
VAR_IN_OUT
	Event			: ST_ErrorStruct;
END_VAR

VAR_IN_OUT CONSTANT
	Monitor			: ST_System_Monitor;
END_VAR

VAR_OUTPUT
	Column				: ARRAY [0..Datalogger.NUMBEROFCOLUMNS] OF ST_Datalog_event; 
END_VAR

VAR
	s_Time				: STRING;
END_VAR
s_Time := SEL(event.b_ErrorActive, event.s_TimeError, event.s_TimeCleared);

Column[0].s_header := 'Date';
Column[0].s_data:= event.s_DateError;

Column[1].s_header := 'Time';
column[1].s_data := s_Time;

Column[2].s_header := 'ID';
column[2].s_data := TO_STRING(event.w_ID);

Column[3].s_header := 'Severity';
column[3].s_data := event.s_Severity;

Column[4].s_header := 'Message';
column[4].s_data := event.s_Message;

Column[5].s_header := 'System state';
column[5].s_data := TO_STRING(monitor.system.e_State);

Column[6].s_header := 'Powerstack state';
column[6].s_data := TO_STRING(monitor.powerstack.e_State);

Column[7].s_header := 'Battery state';
column[7].s_data := TO_STRING(monitor.battery.BatteryInfo.e_BMS_Status);

Column[8].s_header := 'Cooling state';
column[8].s_data := TO_STRING(monitor.Cooling.CoolingSystemMode);

Column[9].s_header := 'Internal Supply Source';
column[9].s_data := TO_STRING(monitor.internalpsu.e_400VSupplySource);

Column[10].s_header := 'Absolute SOC';
column[10].s_data := TO_STRING(monitor.battery.BatteryInfo.r_SOC);

Column[11].s_header := 'DC power';
column[11].s_data := TO_STRING(monitor.battery.BatteryInfo.r_SystemPower);

Column[11].s_header := 'AC apparent power';
column[11].s_data := TO_STRING(monitor.powerstack.r_ApparentPower);
END_METHOD

END_FUNCTION_BLOCK

// ---- POUs/Datalogger/FUNCTIONBLOCKS/FB_CSVWriter.TcPOU
FUNCTION_BLOCK FB_CSVWriter
(* This function block writes comma separated field values to external data buffer *)
VAR_INPUT
	eCmd			: E_EnumCmdType := eEnumCmd_First;(* Command type: write first or next field ?*)
	putValue		: T_MaxString := '';(* New first/next field value as string *)
	pValue			: DWORD := 0;(* OPTIONAL: Pointer to external buffer containing field value data. *)
	cbValue			: UDINT := 0;(* OPTIONAL: Byte size of external buffer containing field value data.  *)
	bCRLF			: BOOL := FALSE;(* TRUE = > Append end of record separator (CR) *)
	bCR				: BOOL := FALSE;(* TRUE = > Append end of record separator (CR) *)
	bLF				: BOOL := FALSE;(* TRUE = > Append end of record separator (LF) *)
	pBuffer  		: PVOID;(* Address ( pointer) of data buffer *)
	cbBuffer		: UDINT;(* Max. byte size of data buffer *)
END_VAR
VAR_OUTPUT
	bOk 			: BOOL;(* TRUE => Successfull, FALSE => Failed *)
	cbSize			: UDINT;(* Number fo used data bytes *)
	cbFree			: UDINT;(* Number of free data bytes *)
	nFields			: UDINT;(* Number of fields *)
	nRecords		: UDINT;(* Number of records *)
	cbWrite			: UDINT;(* Number of successfully written data bytes *)
END_VAR
{library private}
VAR
	fbReader		: FB_CSVMemBufferReader;
	temp			: ARRAY[0..300] OF BYTE;(* Temp buffer *)
	cbTemp			: UDINT := 0;(* Number of data bytes in temp buffer *)
	cbCopied		: UDINT := 0;(* Number of data bytes copied to the external data buffer *)
	bNewLine		: BOOL := TRUE;(* TRUE => start with new line *)
END_VAR

bOk 		:= FALSE;
cbWrite 	:= 0;
(* check external buffer parameter *)
IF ( pBuffer = 0 ) OR ( cbBuffer = 0 ) THEN
	RETURN;
END_IF

(* check pointer and size of binary data *)
IF ( pValue = 0 ) XOR ( cbValue = 0 ) THEN(* Error: One of the parameter is zero and the other one not *)
	RETURN;
ELSE
	cbTemp := MEMCPY( ADR( temp ), ADR( putValue ), MIN( SIZEOF( temp ) - 2, INT_TO_UDINT( LEN( putValue ) ) ) );(* Copy string input data to temp buffer *)
	IF ( pValue <> 0 ) THEN
		IF  ( cbTemp > 0 ) THEN(* Error: Two source inputs: string and buffer are not allowed *)
			RETURN;
		END_IF

		(* binary input => check if the data bytes are enclosed in double-quotation marks *)
		IF cbValue < 2 THEN(* Error: Two double-quotation marks are required! *)
			RETURN;(* Error: Invalid binary input data format *)
		END_IF

		IF ( DWORD_TO_BYTE( pValue)	<> DEFAULT_CSV_FIELD_DOUBLE_QUOTE )						
		OR ( UDINT_TO_BYTE( pValue + cbValue - 1 ) <> DEFAULT_CSV_FIELD_DOUBLE_QUOTE )		
		THEN(* Error: Invalid binary input data format *)                                   
			RETURN; 
		END_IF

		(* Copy binary input data to temp buffer *)
		cbTemp := MEMCPY( ADR( temp ), pValue, MIN( SIZEOF( temp ) - 2, cbValue ) );

	END_IF
END_IF

(* Append CRLF (record termination) *)
temp[ cbTemp ] := DEFAULT_CSV_RECORD_SEP_CR;
temp[ cbTemp + 1 ] := DEFAULT_CSV_RECORD_SEP_LF;
cbTemp := cbTemp + 2;

(* Read and check the new field value *)
fbReader( eCmd := eEnumCmd_First, pBuffer := ADR( temp ), cbBuffer := cbTemp );
IF NOT fbReader.bOk THEN
	RETURN;
END_IF

CASE eCmd OF
	eEnumCmd_First:(* put first field to the buffer => initialize/reset internal variables *)
		bNewLine := TRUE;
		cbSize 		:= 0;
		cbFree 	:= cbBuffer;
		nFields 	:= 0;
		nRecords 	:= 0;
		MEMSET( pBuffer, 0, cbBuffer );(* reset all buffer data bytes *)
	eEnumCmd_Next:(* put next field to the buffer *)
		;(* OK *)
ELSE(* invalid command *)
	RETURN;
END_CASE

(* Check free buffer space *)
IF ( fbReader.cbValue + SEL( bNewLine, 1, 0 ) + SEL( bCRLF, 0, 2 ) ) > cbFree THEN
	RETURN;(* buffer overflow *)
END_IF

(* Write separator (don't write field separator at the beginning of new line) *)
IF bNewLine THEN
	bNewLine := FALSE;
	cbCopied := 0;
ELSE(* copy field separator *)
	cbCopied := MEMSET( pBuffer + cbSize, DEFAULT_CSV_FIELD_SEP, 1 );
END_IF

(* Write field value *)
IF ( fbReader.cbValue > 0 ) AND ( fbReader.pValue <> 0 ) THEN
	cbCopied := cbCopied + MEMCPY( pBuffer + cbSize + cbCopied, fbReader.pValue, fbReader.cbValue );
END_IF
nFields 	:= nFields + 1;

(* Write record termination (CRLF) *)
IF bCRLF THEN
	cbCopied := cbCopied + MEMSET( pBuffer + cbSize + cbCopied, DEFAULT_CSV_RECORD_SEP_CR, 1 );
	cbCopied := cbCopied + MEMSET( pBuffer + cbSize + cbCopied, DEFAULT_CSV_RECORD_SEP_LF, 1 );
	nRecords := nRecords + 1;
	bNewLine := TRUE;
END_IF
IF bCR THEN
	cbCopied := cbCopied + MEMSET( pBuffer + cbSize + cbCopied, DEFAULT_CSV_RECORD_SEP_CR, 1 );
END_IF
IF bLF THEN
	cbCopied := cbCopied + MEMSET( pBuffer + cbSize + cbCopied, DEFAULT_CSV_RECORD_SEP_LF, 1 );
	nRecords := nRecords + 1;
	bNewLine := TRUE;
END_IF

cbSize 		:= cbSize + cbCopied;
cbFree		:= cbBuffer - cbSize;
cbWrite	:= cbCopied;
bOk 		:= TRUE;

END_FUNCTION_BLOCK

// ---- POUs/Datalogger/FUNCTIONBLOCKS/ToHexConverter.TcPOU
FUNCTION_BLOCK ToHexConverter
VAR_INPUT
	var1 : BOOL;
	var2 : BOOL;
	var3 : BOOL;
	var4 : BOOL;
	var5 : BOOL;
	var6 : BOOL;
	var7 : BOOL;
	var8 : BOOL;
END_VAR
VAR_OUTPUT
	Stringtotal : STRING;
END_VAR
VAR
	BTOT14 : INT;
	BTOT58 : INT;
	ivar1 : INT;
	ivar2 : INT;
	ivar3 : INT;
	ivar4 : INT;
	ivar5 : INT;
	ivar6 : INT;
	ivar7 : INT;
	ivar8 : INT;
	String1 : STRING;
	String2 : STRING;
END_VAR

ivar1 := BOOL_TO_INT(var1);
ivar2 := BOOL_TO_INT(var2);
ivar3 := BOOL_TO_INT(var3);
ivar4 := BOOL_TO_INT(var4);
ivar5 := BOOL_TO_INT(var5);
ivar6 := BOOL_TO_INT(var6);
ivar7 := BOOL_TO_INT(var7);
ivar8 := BOOL_TO_INT(var8);

iVar1 := ivar1 * 8;
iVar2 := ivar2 * 4;
iVar3 := ivar3 * 2;
iVar4 := ivar4 * 1;

iVAR5 := ivar5 * 8;
iVar6 := ivar6 * 4;
iVar7 := ivar7 * 2;
iVar8 := ivar8 * 1;

BTOT14 := iVar1 + iVar2 + iVar3 + iVar4;

BTOT58 := iVar5 + iVar6 + iVar7 + iVar8;
 
IF BTOT14 = 10 THEN 
	String1 := 'A';
ELSE IF BTOT14 = 11 THEN 
	String1 := 'B';
ELSE IF BTOT14 = 12 THEN 
	String1 := 'C';
ELSE IF BTOT14 = 13 THEN 
	String1 := 'D';
ELSE IF BTOT14 = 14 THEN 
	String1 := 'E';
ELSE IF BTOT14 = 15 THEN 
	String1 := 'F';
ELSE
	String1 := INT_TO_STRING(BTOT14);
END_IF
END_IF
END_IF
END_IF
END_IF
END_IF

IF BTOT58 = 10 THEN 
	String2 := 'A';
ELSE IF BTOT58 = 11 THEN 
	String2 := 'B';
ELSE IF BTOT58 = 12 THEN 
	String2 := 'C';
ELSE IF BTOT58 = 13 THEN 
	String2 := 'D';
ELSE IF BTOT58 = 14 THEN 
	String2 := 'E';
ELSE IF BTOT58 = 15 THEN 
	String2 := 'F';
ELSE
	String2 := INT_TO_STRING(BTOT58);
END_IF
END_IF
END_IF
END_IF
END_IF
END_IF

StringTotal := CONCAT( String1, String2);

END_FUNCTION_BLOCK

// ---- POUs/EventLogger/EventLog.TcPOU
PROGRAM EventLog


VAR
	WriteTest		:	BOOL;
	fbOpenFile 		: FB_Fileopen;
	fbWriteFile		: FB_FilePuts;
	fbCloseFile 	: FB_FileClose;
	fbRenameFile	: FB_FileRename;
	fbDeleteFile	: FB_FileDelete;
	fbFileInfo		:	FB_EnumFindFileEntry;
	stFiledata		:	ST_FindFileEntry;
	FileOpenDone		:	F_TRIG;
	FileWriteDone		:	F_TRIG;
	FileCloseDone		:	F_TRIG;
	FileRenameDone		:	F_TRIG;
	FileDeleteDone		:	F_TRIG;
	FileInfoDone		:	F_TRIG;
	FileSize			:	ULINT;
	FileCounter			:	INT;
	Filehandle 			: UINT;
	
	bForceWrite 			:	BOOL;	//immediately flush out buffer on shutdown
	bEMstopWrite			:	BOOL;	//Flush out after EMStop, but give some time for final logs to come in 
	tonEMstopDelay			:	TON;
	tonGeneralWriteDelay	:	Ton;
	FileActionDelay			:	TON := (PT := T#30MS);

	MemoryBuffer	:	FB_StringRingBuffer;
	DataBuffer		:	ARRAY[0..100000] OF BYTE; //100kb to start
	WriteString	:	t_MAXSTRING;

	
	
	Stop_logging	:	Bool;
	
END_VAR

VAR_IN_OUT CONSTANT
	STParams : ST_EventLoggerParams;
END_VAR

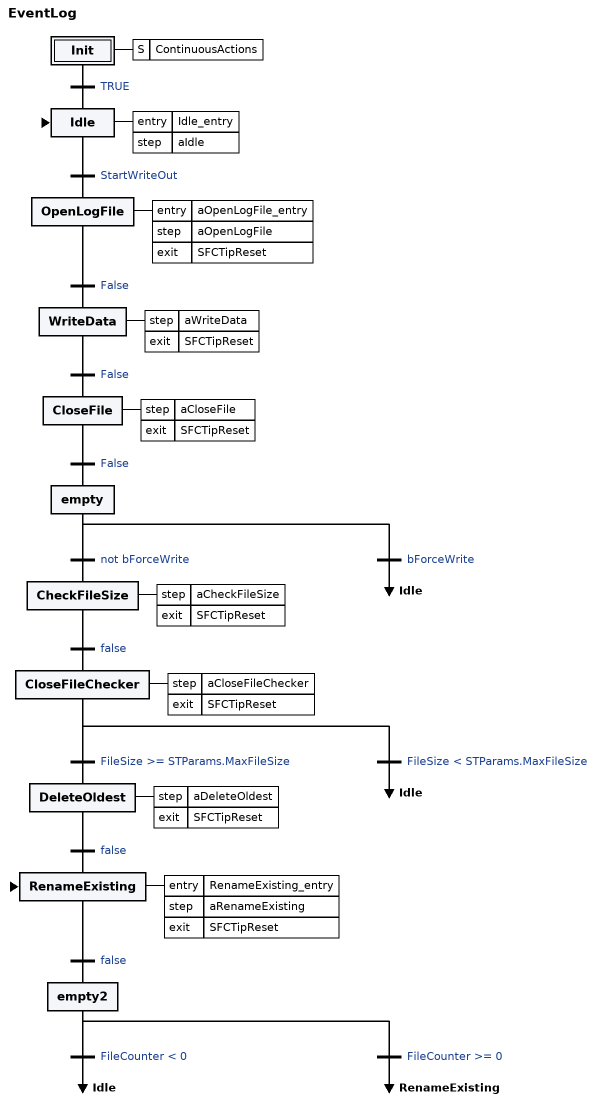
INITIAL_STEP Init:
    ContinuousActions(S);
END_STEP
TRANSITION FROM Init TO Idle
    := TRUE;
END_TRANSITION
STEP Idle:
    Idle_entry(P1);  // entry action
    aIdle(N);  // step action
END_STEP
TRANSITION FROM Idle TO OpenLogFile
    := StartWriteOut;
END_TRANSITION
// macro Writeout begins
STEP OpenLogFile:
    aOpenLogFile_entry(P1);  // entry action
    aOpenLogFile(N);  // step action
    SFCTipReset(P0);  // exit action
END_STEP
TRANSITION FROM OpenLogFile TO WriteData
    := False;
END_TRANSITION
STEP WriteData:
    aWriteData(N);  // step action
    SFCTipReset(P0);  // exit action
END_STEP
TRANSITION FROM WriteData TO CloseFile
    := False;
END_TRANSITION
STEP CloseFile:
    aCloseFile(N);  // step action
    SFCTipReset(P0);  // exit action
END_STEP
TRANSITION FROM CloseFile TO empty
    := False;
END_TRANSITION
STEP empty:
END_STEP
TRANSITION FROM empty TO CheckFileSize
    := not bForceWrite;
END_TRANSITION
TRANSITION FROM empty TO Idle
    := bForceWrite;
END_TRANSITION
// macro LogRotate begins
STEP CheckFileSize:
    aCheckFileSize(N);  // step action
    SFCTipReset(P0);  // exit action
END_STEP
TRANSITION FROM CheckFileSize TO CloseFileChecker
    := false;
END_TRANSITION
STEP CloseFileChecker:
    aCloseFileChecker(N);  // step action
    SFCTipReset(P0);  // exit action
END_STEP
TRANSITION FROM CloseFileChecker TO DeleteOldest
    := FileSize >= STParams.MaxFileSize;
END_TRANSITION
STEP DeleteOldest:
    aDeleteOldest(N);  // step action
    SFCTipReset(P0);  // exit action
END_STEP
TRANSITION FROM DeleteOldest TO RenameExisting
    := false;
END_TRANSITION
STEP RenameExisting:
    RenameExisting_entry(P1);  // entry action
    aRenameExisting(N);  // step action
    SFCTipReset(P0);  // exit action
END_STEP
TRANSITION FROM RenameExisting TO empty2
    := false;
END_TRANSITION
STEP empty2:
END_STEP
TRANSITION FROM empty2 TO Idle
    := FileCounter < 0;
END_TRANSITION
TRANSITION FROM empty2 TO RenameExisting
    := FileCounter >= 0;
END_TRANSITION
TRANSITION FROM CloseFileChecker TO Idle
    := FileSize < STParams.MaxFileSize;
END_TRANSITION

ACTION aCheckFileSize:


FileInfoDone(clk := fbFileInfo.bbusy);
FileActionDelay(in:= NOT (fbFileInfo.bbusy OR FileInfoDone.Q));

fbFileInfo(sPathname:= Stparams.LogFileName,
		bExecute := FileActionDelay.Q,
		eCMD := eEnumCmd_First,
		tTimeout := T#100MS);


IF FileInfoDone.q THEN
	FileSize := 0;
	IF NOT fbFileInfo.bError THEN
		IF NOT fbfileInfo.bEOE THEN
			stFiledata := fbFileinfo.stFindFile;
			FileSize := ULARGE_TO_ULINT(stFiledata.fileSize);
		END_IF
	END_IF
	SFCTip := TRUE;
END_IF
END_ACTION

ACTION aCloseFile:

FileCloseDone(clk := fbCloseFile.bbusy);

FileActionDelay(in := NOT (fbCloseFile.bbusy OR FileCloseDone.Q));


fbCloseFile(Hfile := FileHandle,
		bExecute   := FileActionDelay.q,
    	tTimeout   := T#100MS);


IF FileCloseDone.q THEN
	IF NOT fbCloseFile.bError THEN
		filehandle := 0;
		SFCTip := TRUE;
	END_IF
END_IF
END_ACTION

ACTION aCloseFileChecker:


FileInfoDone(clk := fbFileInfo.bbusy);
FileActionDelay(in:= not (fbFileInfo.bbusy OR FileInfoDone.Q));

fbFileInfo(sPathname:= Stparams.LogFileName,
		bExecute := FileActionDelay.Q,
		eCMD := eEnumCmd_Abort,
		tTimeout := T#100MS);


IF FileInfoDone.q THEN
	FileSize := 0;
	IF NOT fbFileInfo.bError THEN
		SFCTip := TRUE;
	END_IF
END_IF
END_ACTION

METHOD AddEvent : BOOL
VAR_INPUT
	LogMessage	:	STRING;
END_VAR
IF NOT Stop_logging THEN	
	MemoryBuffer.A_AddTail(putValue := LogMessage);
end_if
END_METHOD

ACTION aDeleteOldest:

FileDeleteDone(clk := fbDeleteFile.bbusy);
FileActionDelay(in:=NOT (fbDeleteFile.bbusy OR FileDeleteDone.Q));
	
fbDeleteFile(sPathname:= concat(concat(Stparams.LogFileName, '.'),TO_STRING(stparams.MaxFileCount-1)),
		bExecute := FileActionDelay.q,
		tTimeout := T#100MS);


IF FileDeleteDone.q THEN
	//could end in error if file doesn't exist. This is fine.
	FileCounter := stparams.MaxFileCount-2;
	SFCTip := TRUE;
END_IF
END_ACTION

ACTION aIdle:
tonGeneralWriteDelay.IN := true;
END_ACTION

ACTION aOpenLogFile:
bEMStopWrite := FALSE;
tonGeneralWriteDelay.IN := FALSE;
FileOpenDone(clk := fbOpenFile.bbusy);

FileActionDelay(in := NOT (fbOpenFile.bbusy OR FileOpenDone.Q));

fbOpenFile(sPathName := Stparams.LogFileName,
		nMode := FOPEN_MODEAPPEND OR FOPEN_MODETEXT,
		bExecute   :=  FileActionDelay.Q,
    	tTimeout   := T#100MS);


IF FileOpenDone.q THEN
	FileHandle := fbOpenFile.hFile;
	IF FileHandle <> 0 THEN
		MemoryBuffer.A_RemoveHead(getValue => WriteString);
		SFCTip := TRUE;
	END_IF
END_IF
END_ACTION

ACTION aOpenLogFile_entry:

END_ACTION

ACTION aRenameExisting:

FileRenameDone(clk := fbRenameFile.bbusy);
FileActionDelay(in:= NOT (fbDeleteFile.bbusy OR FileDeleteDone.Q));

fbRenameFile(
		bExecute := FileActionDelay.Q,
		tTimeout := T#100MS);


IF FileRenameDone.q THEN
	//could end in error if file doesn't exist. This is fine.
	FileCounter := FileCounter-1;
	SFCTip := TRUE;
END_IF
END_ACTION

ACTION aWriteData:

//add entry action with initial Writestring fill
filehandle;

FileWriteDone(clk := fbWriteFile.bbusy);

FileActionDelay(in := NOT (fbWriteFile.bbusy OR FileWriteDone.Q));

fbWriteFile(hfile := filehandle,
			sLine := WriteString,
			BExecute := FileActionDelay.Q,
			tTimeout := T#500MS);


IF FileWriteDone.q THEN
	IF MemoryBuffer.nCount > 0 THEN //Still data present, continue writing
		MemoryBuffer.A_RemoveHead(getValue => WriteString);
	ELSE //file not opened, back to start?
		SFCTip := TRUE;
	END_IF
END_IF
END_ACTION

ACTION ContinuousActions:
MemoryBuffer(bOverwrite := TRUE, pBuffer := ADR(DataBuffer), cbBuffer := SIZEOF(DataBuffer));
tonEMstopDelay(in := bEMstopWrite, pt:= stparams.EMstopWriteDelay);
tonGeneralWriteDelay(in:= MemoryBuffer.nCount > 0, Pt:=stparams.LogWriteInterval);

IF WriteTest THEN
	WriteLogItem(Source := eObject_ID.System, Severity := eSeverity.Warning, LogText := 'testtesttest');
	WriteTest := FALSE;
	bEMstopWrite := TRUE;
END_IF
END_ACTION

METHOD EMstop : BOOL
VAR_INPUT
END_VAR

VAR
	LogText	:	String;
END_VAR

IF memorybuffer.nCount > 0 THEN
	bEMstopWrite := TRUE;
END_IF

EMStop := TRUE;
END_METHOD

ACTION Idle_entry:
bEMStopWrite := FALSE;
bForceWrite := FALSE;
END_ACTION

ACTION RenameExisting_entry:

IF FileCounter = 0 THEN 
	fbRenameFile.sOldName := Stparams.LogFileName;
ELSE
	fbRenameFile.sOldName := concat(concat(Stparams.LogFileName, '.'),TO_STRING(FileCounter));
END_IF
fbRenameFile.sNewName	:= concat(concat(Stparams.LogFileName, '.'),TO_STRING(FileCounter+1));
END_ACTION

ACTION SFCTipReset:
FileActionDelay(in := FALSE);
SFCTip := false;
END_ACTION

METHOD Shutdown : BOOL
VAR_INPUT
END_VAR

IF memorybuffer.nCount > 0 THEN
	bForceWrite := TRUE;
END_IF

Shutdown := TRUE;
END_METHOD

TRANSITION StartWriteOut:
//Flush logs to file if
MemoryBuffer.cbSize > TO_UDINT(stparams.MaxFillGrade*MemoryBuffer.cbBuffer) OR //buffer gets full
tonGeneralWriteDelay.Q  OR //fixed interval
tonEmstopDelay.Q OR //just after emstop
bForceWrite; //at systemshutdown
END_TRANSITION

END_PROGRAM

// ---- POUs/EventLogger/WriteLogItem.TcPOU
FUNCTION WriteLogItem : Bool
VAR_INPUT
	Source		: eObject_ID;
	Severity	: eSeverity;
	LogText		: STRING(200);
END_VAR

VAR
	LogString	:	STRING(255);
END_VAR


Logstring := CONCAT(DT_TO_STRING(GVL.dt_SystemDateTime), ' - ');//20 char?
Logstring := CONCAT(Logstring, TO_STRING(Source));				//19 char
Logstring := CONCAT(Logstring, ' - ');							//3 char
Logstring := CONCAT(Logstring, TO_STRING(Severity));			//7 char
Logstring := CONCAT(Logstring, ' - ');							//3 char
Logstring := CONCAT(Logstring, LogText);
Logstring := CONCAT(Logstring, '$0A');							//1 char

EventLog.AddEvent(LogString);

END_FUNCTION

// ---- POUs/Functions-FBs-Programs/FB_OverCurrentDetect.TcPOU
FUNCTION_BLOCK FB_OverCurrentDetect
VAR_INPUT
	ui_Ik					: UINT := 10; // kA/s 
	ui_RatedCurrent			: UINT; // A
	ui_gain					: UINT := 15;
	b_reset					: BOOL;
	r_In					: REAL;
	t_ResetTime				: TIME := T#2S;  
	t_MaxPickUpTime			: TIME := T#30M;
END_VAR
	
VAR_OUTPUT
	b_alarm						: BOOL;
	b_warning					: BOOL;
	ui_actLoad					: UINT; //%
	r_MaxCurrentDetected		: REAL;
	t_MaxTimeActive				: TIME;
	t_RemainingTime				: TIME;
END_VAR
VAR
	ton_PickUpTimer			: TON := (PT:=T#10S);
	ton_ResetTimer			: TON := (PT:=T#5S);
	r_MaxCurrent			: REAL;
	t_MaxTime				: TIME;
END_VAR

VAR
	r_ThermalMax		 	: REAL ;
	r_CurrentLimit			: REAL;
	r_Overcurrent			: REAL;
	r_thermalLoad			: REAL;
	r_thermalDelta			: REAL;
	r_thermalEnergy			: REAL;
	r_StepSize				: REAL;				
	//fb_loadMa				: FB_MovingAverage := (enable:= TRUE);
	i_instance				: INT;	
	init					: BOOL := TRUE;	
END_VAR

VAR_STAT
	i_instanceCounter		: INT;
	ton_evalTimer			: TON := (PT := T#10MS);
END_VAR

ton_pickUpTimer(PT:=t_MaxPickUpTime);
ton_ResetTimer(PT:=t_ResetTime);


IF i_instance = 0 THEN
	ton_EvalTimer(IN := NOT ton_evaltimer.Q);
END_IF

IF ton_evalTimer.Q THEN
	r_thermalMax := EXPT(TO_REAL(ui_Ik) * 1000,2);
	r_CurrentLimit := TO_REAL(ui_ratedCurrent);
	r_OverCurrent := r_in - r_CurrentLimit ;
	r_thermalLoad := EXPT(r_in, 2);
	r_StepSize := TO_REAL(ton_evalTimer.PT) / 1000;
	r_thermalDelta := EXPT(r_overcurrent * SEL(r_OverCurrent >0, ui_gain / 5, ui_gain),2) * SEL(r_OverCurrent >0, -1, 1);
	r_thermalEnergy := LIMIT(0, r_thermalEnergy + r_ThermalDelta * r_stepsize * 2, r_thermalMax * 1.01); // unknown why *2, but this gives correct remaining time...

	//fb_loadMa(IN := MAX(0,r_thermalDelta), Length := 2);
	
	IF r_IN >= r_CurrentLimit THEN
		t_remainingTime := MIN(t_maxPickUpTime - ton_pickUpTimer.ET, TO_TIME((MAX(0,r_thermalMax - r_thermalEnergy)) / MAX(1, r_thermalDelta) *1000)); 
		ui_actLoad := TO_UINT(r_In / MAX(1,ui_RatedCurrent) * 100);
		ton_PickUpTimer.IN := TRUE;
		ton_ResetTimer.IN := FALSE;
		IF t_MaxTime < ton_PickUpTimer.ET THEN
			t_MaxTime := ton_PickUpTimer.ET;
			t_MaxTimeActive := t_MaxTime;
		END_IF
		
		IF r_MaxCurrent < ABS(r_IN) THEN
			r_MaxCurrent := ABS(r_IN);
			r_MaxCurrentDetected := r_MaxCurrent;
		END_IF
	ELSIF r_IN < r_CurrentLimit THEN
		t_remainingTime := t_MaxPickUpTime;
		ton_ResetTimer.IN := TRUE;
		ton_PickUpTimer.IN := NOT(ton_ResetTimer.Q);
	END_IF
	
	b_Alarm := ton_PickUpTimer.Q OR t_remainingTime = T#0S;
	b_Warning := ton_PickUpTimer.IN;
	
	IF NOT ton_PickUpTimer.IN THEN
		ui_actLoad := 0;
		r_maxCurrent := 0;
		t_MaxTime := T#0S;
	END_IF
	
	IF b_reset THEN
		r_thermalEnergy := 0;
		r_MaxCurrentDetected := 0;
		t_MaxTimeActive := T#0S;
	END_IF

END_IF


IF init THEN
	init := FALSE;
	i_instance := i_instanceCounter;
	i_instanceCounter:= i_instanceCounter +1;
END_IF

END_FUNCTION_BLOCK

// ---- POUs/Functions-FBs-Programs/FB_UpperLimitAndTimeExceeded.TcPOU
FUNCTION_BLOCK FB_UpperLimitAndTimeExceeded
VAR_INPUT
	b_reset					: BOOL;
	r_In					: REAL;
	r_HighLimit				: REAL;
	r_Hysteresis			: REAL := 10;
	t_ResetTIME				: TIME;  
	t_PickUpTime			: TIME;
END_VAR
	
VAR_OUTPUT
	b_alarm						: BOOL;
	b_warning					: BOOL;
	r_MaxCurrentDetected		: REAL;
	t_MaxTimeActive				: TIME;
END_VAR
VAR
	ton_PickUpTimer			: TON := (PT:=T#10S);
	ton_ResetTimer			: TON := (PT:=T#5S);
	r_MaxCurrent			: REAL;
	t_MaxTime				: TIME;
END_VAR

ton_pickUpTimer(PT:=t_PickUpTime);
ton_ResetTimer(PT:=t_ResetTime);

IF r_IN >= r_HighLimit THEN
	ton_PickUpTimer.IN := TRUE;
	ton_ResetTimer.IN := FALSE;
	IF t_MaxTime < ton_PickUpTimer.ET THEN
		t_MaxTime := ton_PickUpTimer.ET;
		t_MaxTimeActive := t_MaxTime;
	END_IF
	
	IF r_MaxCurrent < ABS(r_IN) THEN
		r_MaxCurrent := ABS(r_IN);
		r_MaxCurrentDetected := r_MaxCurrent;
	END_IF
ELSIF r_IN < (r_HighLimit - r_Hysteresis) THEN
	ton_ResetTimer.IN := TRUE;
	ton_PickUpTimer.IN := NOT(ton_ResetTimer.Q);
END_IF

b_Alarm := ton_PickUpTimer.Q;
b_Warning := ton_PickUpTimer.IN;

IF NOT ton_PickUpTimer.IN THEN
	r_maxCurrent := 0;
	t_MaxTime := T#0S;
END_IF

IF b_reset THEN
	r_MaxCurrentDetected := 0;
	t_MaxTimeActive := T#0S;
END_IF

END_FUNCTION_BLOCK

// ---- POUs/Functions-FBs-Programs/_generalFunctions/PackByte.TcPOU
FUNCTION PackByte : INT
VAR_INPUT
	B0				: BOOL ;
	B1				: BOOL ;
	B2				: BOOL ;
	B3				: BOOL ;
	B4				: BOOL ;
	B5				: BOOL ;
	B6				: BOOL ;
	B7				: BOOL ;	
END_VAR
VAR
END_VAR

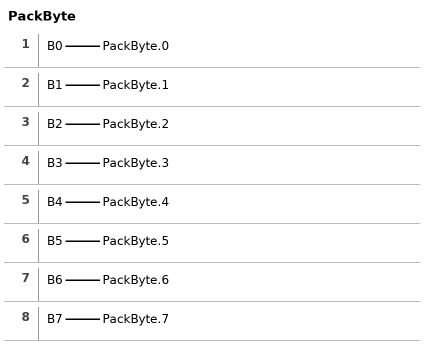
// NETWORK 1
PackByte.0 := B0;

// NETWORK 2
PackByte.1 := B1;

// NETWORK 3
PackByte.2 := B2;

// NETWORK 4
PackByte.3 := B3;

// NETWORK 5
PackByte.4 := B4;

// NETWORK 6
PackByte.5 := B5;

// NETWORK 7
PackByte.6 := B6;

// NETWORK 8
PackByte.7 := B7;

END_FUNCTION

// ---- POUs/Functions-FBs-Programs/_generalFunctions/XNOR.TcPOU
FUNCTION XNOR : BOOL
VAR_INPUT
	a : BOOL;
	b : BOOL;
END_VAR
VAR
END_VAR

XNOR := a AND b OR NOT (a OR b);

END_FUNCTION

// ---- POUs/Objects/InterMachineCom/FB_ConnectMqttBroker.TcPOU
FUNCTION_BLOCK FB_ConnectMqttBroker
VAR_INPUT
	bRestartConnection			: BOOL;
	bConnect					: BOOL;
	sHostName					: STRING;
					
END_VAR
VAR_OUTPUT
	eConnectionState			: eConnectionState;
	bIncomingMsg	: BOOL;
	sMessage		: STRING;
END_VAR
VAR
	fbMqttClient					: FB_IotMqttClient;
	fbMessageQueue					: FB_IotMqttMessageQueue;
	fbMessage						: FB_IotMqttMessage;
	ton_ReconnectionTimer			: TON := (PT:=T#5S);
	bSetParameter					: BOOL;
	rTrigReinitCom					: R_TRIG;
	rTrigComStateOK					: R_Trig;
	
	//subscription
	bSubscribed 					: BOOL;
	sSubscribedTopic 				: STRING;
	sReceivedTopic					: STRING;
	
	//json files
	fbJson         	: FB_JsonSaxWriter;
  	fbJsonDataType 	: FB_JsonReadWriteDataType;
	sJsonDocPub     : STRING(255);
END_VAR

ton_ReconnectionTimer(IN:= NOT ton_ReConnectionTimer.Q AND NOT fbMqttClient.bConnected);
rTrigReinitCom(CLK := bRestartConnection);
bIncomingMsg := FALSE;

IF ton_reconnectionTimer.Q OR rTrigReinitCom.Q THEN
	eConnectionState := eConnectionState.disconnected;
	//Reset connection
	fbMqttClient.Execute(FALSE);
	//Configure
	IF bSetParameter THEN
		bSetParameter := FALSE;
		fbMqttClient.sHostName							:= sHostName;
		fbMqttClient.nHostPort							:= 1883;
		fbMqttClient.ipMessageQueue						:= fbMessageQueue;
	END_IF
ELSE
	fbMqttClient.Execute(bConnect);
	//Reset parameter set for next time connecting
	bSetParameter := TRUE;
END_IF

rTrigComStateOK(CLK := fbMqttClient.bConnected);
IF rTrigComStateOK.Q THEN
	eConnectionState := eConnectionState.connected;
END_IF


//receive message at subscribed topic
IF fbMessageQueue.nQueuedMessages > 0 THEN
	 IF fbMessageQueue.Dequeue(fbMessage:=fbMessage) THEN
		fbMessage.GetTopic(pTopic:=ADR(sReceivedTopic), nTopicSize:=SIZEOF(sReceivedTopic) );
			// Process asset messages
			bIncomingMsg	:= TRUE;
			fbMessage.GetPayload(pPayload:=ADR(sMessage), nPayloadSize:=SIZEOF(sMessage), bSetNullTermination:=TRUE);
			sMessage:=LEFT(sMessage,LEN(sMessage) -1 );
	END_IF
END_IF

//TO ADD, when no slaves are present, reduce publish interval

METHOD Publish : BOOL
VAR_INPUT
	Interval		: TIME;
	sTopic			: STRING;
	sMessage		: STRING;
END_VAR

VAR_INST
	tMinInterval 				: TIME := T#10MS;
	tonPublishInterval			: TON;
END_VAR
// publish
tonpublishInterval(PT := MAX(tMinInterval, Interval));

IF fbMqttClient.bConnected THEN
    tonPublishInterval.IN := TRUE;
    IF tonPublishInterval.Q THEN // publish new payload every second
        tonPublishInterval.IN := FALSE;
		fbMqttClient.Publish(sTopic:=sTopic,
		pPayload := ADR(sMessage),
		nPayloadSize := LEN2(ADR(sMessage)),
		eQoS := TcIotMqttQos.AtMostOnceDelivery,
		bRetain:= FALSE,
		bQueue := FALSE);
    END_IF
END_IF
END_METHOD

METHOD Subscribe : BOOL;
VAR_INPUT
	sTopic		: STRING; 
END_VAR

VAR_INST
	sReceivedTopic : STRING;
END_VAR
IF fbMqttClient.bConnected AND NOT bSubscribed THEN
	sSubscribedTopic := sTopic;
   bSubscribed := fbMqttClient.Subscribe(sTopic:=sTopic, eQoS:=TcIotMqttQos.AtMostOnceDelivery); //sSubTopic
END_IF

IF sSubscribedTopic <> sTopic THEN
	bSubscribed := FALSE;
END_IF
END_METHOD

END_FUNCTION_BLOCK

// ---- POUs/Objects/InterMachineCom/FB_InterMachineCommunication.TcPOU
FUNCTION_BLOCK FB_InterMachineCommunication
VAR_INPUT
	SlaveConnectionData				: ST_InterMachineCom_SlaveConData;

END_VAR

VAR_IN_OUT CONSTANT
	monitor							: ST_system_monitor;
	st_params						: ST_InterMachineCom_Params;
END_VAR

VAR_IN_OUT
	control							: ST_system_control;
END_VAR

VAR_OUTPUT
	e_state							: eConnectionState;
END_VAR

VAR
	InternalBroker					: FB_ConnectMqttBroker;
	ExternalBroker					: FB_ConnectMQttBroker;
	
